LIN {X 0,Y 192.348,Z 460.48,A -85,B 0,C 180,E1 -21860.529,E2 -21860.529} C_VEL
LIN {X 0,Y 193.959,Z 454.471,A -85,B 0,C 180,E1 -21863.761,E2 -21863.761} C_VEL
LIN {X 0,Y 196.232,Z 446.608,A -85,B 0,C 180,E1 -21867.025,E2 -21867.025} C_VEL
LIN {X 0,Y 198.774,Z 437.463,A -85,B 0,C 180,E1 -21870.002,E2 -21870.002} C_VEL
LIN {X 0,Y 201.367,Z 427.594,A -85,B 0,C 180,E1 -21872.502,E2 -21872.502} C_VEL
LIN {X 0,Y 204.103,Z 416.202,A -85,B 0,C 180,E1 -21874.764,E2 -21874.764} C_VEL
LIN {X 0,Y 206.217,Z 405.922,A -85,B 0,C 180,E1 -21876.361,E2 -21876.361} C_VEL
LIN {X 0,Y 208.161,Z 394.258,A -85,B 0,C 180,E1 -21877.763,E2 -21877.763} C_VEL
LIN {X 0,Y 209.919,Z 381.041,A -85,B 0,C 180,E1 -21878.909,E2 -21878.909} C_VEL
LIN {X 0,Y 211.115,Z 368.346,A -85,B 0,C 180,E1 -21879.633,E2 -21879.633} C_VEL
LIN {X 0,Y 213.846,Z 309.716,A -85,B 0,C 180,E1 -21881.608,E2 -21881.608} C_VEL
LIN {X 0,Y 206.528,Z 290.704,A -85,B 0,C 180,E1 -21883.594,E2 -21883.594} C_VEL
LIN {X 0,Y 198.591,Z 273.838,A -85,B 0,C 180,E1 -21885.769,E2 -21885.769} C_VEL
LIN {X 0,Y 194.153,Z 266.401,A -85,B 0,C 180,E1 -21886.995,E2 -21886.995} C_VEL
LIN {X 0,Y 192.896,Z 263.787,A -85,B 0,C 180,E1 -21887.477,E2 -21887.477} C_VEL
LIN {X 0,Y 192.743,Z 263.034,A -85,B 0,C 180,E1 -21887.926,E2 -21887.926} C_VEL
LIN {X 0,Y 192.652,Z 262.975,A -85,B 0,C 180,E1 -21893.66,E2 -21893.66} C_VEL
LIN {X 0,Y 192.577,Z 262.979,A -85,B 0,C 180,E1 -21898.87,E2 -21898.87} C_VEL
LIN {X 0,Y 192.571,Z 262.99,A -85,B 0,C 180,E1 -21903.193,E2 -21903.193} C_VEL
LIN {X 0,Y 192.521,Z 263.004,A -85,B 0,C 180,E1 -21908.361,E2 -21908.361} C_VEL
LIN {X 0,Y 192.465,Z 262.982,A -85,B 0,C 180,E1 -21913.1,E2 -21913.1} C_VEL
LIN {X 0,Y 192.469,Z 263.011,A -85,B 0,C 180,E1 -21916.913,E2 -21916.913} C_VEL
LIN {X 0,Y 192.527,Z 262.965,A -85,B 0,C 180,E1 -21921.653,E2 -21921.653} C_VEL
LIN {X 0,Y 192.583,Z 262.994,A -85,B 0,C 180,E1 -21926.821,E2 -21926.821} C_VEL
LIN {X 0,Y 192.601,Z 262.948,A -85,B 0,C 180,E1 -21931.691,E2 -21931.691} C_VEL
LIN {X 0,Y 192.653,Z 262.986,A -85,B 0,C 180,E1 -21936.35,E2 -21936.35} C_VEL
LIN {X 0,Y 192.692,Z 262.933,A -85,B 0,C 180,E1 -21941.498,E2 -21941.498} C_VEL
LIN {X 0,Y 192.739,Z 262.95,A -85,B 0,C 180,E1 -21945.22,E2 -21945.22} C_VEL
LIN {X 0,Y 192.946,Z 262.944,A -85,B 0,C 180,E1 -21949.574,E2 -21949.574} C_VEL
LIN {X 0,Y 192.965,Z 262.897,A -85,B 0,C 180,E1 -21953.735,E2 -21953.735} C_VEL
LIN {X 0,Y 193.232,Z 262.904,A -85,B 0,C 180,E1 -21957.923,E2 -21957.923} C_VEL
LIN {X 0,Y 193.417,Z 262.891,A -85,B 0,C 180,E1 -21960.007,E2 -21960.007} C_VEL
LIN {X 0,Y 192.937,Z 262.907,A -85,B 0,C 180,E1 -21964.185,E2 -21964.185} C_VEL
LIN {X 0,Y 193.039,Z 262.926,A -85,B 0,C 180,E1 -21968.381,E2 -21968.381} C_VEL
LIN {X 0,Y 192.805,Z 262.955,A -85,B 0,C 180,E1 -21972.64,E2 -21972.64} C_VEL
LIN {X 0,Y 192.732,Z 262.949,A -85,B 0,C 180,E1 -21976.968,E2 -21976.968} C_VEL
LIN {X 0,Y 192.62,Z 262.984,A -85,B 0,C 180,E1 -21981.406,E2 -21981.406} C_VEL
LIN {X 0,Y 192.652,Z 262.956,A -85,B 0,C 180,E1 -21984.213,E2 -21984.213} C_VEL
LIN {X 0,Y 192.616,Z 262.987,A -85,B 0,C 180,E1 -21988.87,E2 -21988.87} C_VEL
LIN {X 0,Y 192.609,Z 262.983,A -85,B 0,C 180,E1 -21993.191,E2 -21993.191} C_VEL
LIN {X 0,Y 192.557,Z 262.985,A -85,B 0,C 180,E1 -21998.358,E2 -21998.358} C_VEL
LIN {X 0,Y 192.5,Z 262.993,A -85,B 0,C 180,E1 -22003.096,E2 -22003.096} C_VEL
LIN {X 0,Y 192.598,Z 263.215,A -85,B 0,C 180,E1 -22007.845,E2 -22007.845} C_VEL
LIN {X 0,Y 193.472,Z 266.459,A -85,B 0,C 180,E1 -22009.626,E2 -22009.626} C_VEL
LIN {X 0,Y 199.825,Z 279.379,A -85,B 0,C 180,E1 -22011.546,E2 -22011.546} C_VEL
LIN {X 0,Y 207.254,Z 296.355,A -85,B 0,C 180,E1 -22013.6,E2 -22013.6} C_VEL
LIN {X 0,Y 212.281,Z 309.796,A -85,B 0,C 180,E1 -22014.982,E2 -22014.982} C_VEL
LIN {X 0,Y 213.59,Z 320.418,A -85,B 0,C 180,E1 -22015.614,E2 -22015.614} C_VEL
LIN {X 0,Y 213.361,Z 326.003,A -85,B 0,C 180,E1 -22015.803,E2 -22015.803} C_VEL
LIN {X 0,Y 212.523,Z 331.839,A -85,B 0,C 180,E1 -22015.909,E2 -22015.909} C_VEL
LIN {X 0,Y 206.506,Z 350.757,A -85,B 0,C 180,E1 -22015.752,E2 -22015.752} C_VEL
LIN {X 0,Y 205.647,Z 356.594,A -85,B 0,C 180,E1 -22015.859,E2 -22015.859} C_VEL
LIN {X 0,Y 204.571,Z 375.827,A -85,B 0,C 180,E1 -22016.577,E2 -22016.577} C_VEL
LIN {X 0,Y 203.127,Z 389.153,A -85,B 0,C 180,E1 -22017.42,E2 -22017.42} C_VEL
LIN {X 0,Y 201.302,Z 401.297,A -85,B 0,C 180,E1 -22018.565,E2 -22018.565} C_VEL
LIN {X 0,Y 199.045,Z 413.08,A -85,B 0,C 180,E1 -22020.082,E2 -22020.082} C_VEL
LIN {X 0,Y 196.366,Z 424.446,A -85,B 0,C 180,E1 -22021.98,E2 -22021.98} C_VEL
LIN {X 0,Y 193.702,Z 434.702,A -85,B 0,C 180,E1 -22024.188,E2 -22024.188} C_VEL
LIN {X 0,Y 191.305,Z 443.865,A -85,B 0,C 180,E1 -22026.711,E2 -22026.711} C_VEL
LIN {X 0,Y 189.106,Z 451.549,A -85,B 0,C 180,E1 -22029.324,E2 -22029.324} C_VEL
LIN {X 0,Y 186.872,Z 458.998,A -85,B 0,C 180,E1 -22032.488,E2 -22032.488} C_VEL
LIN {X 0,Y 185.181,Z 464.964,A -85,B 0,C 180,E1 -22035.717,E2 -22035.717} C_VEL
LIN {X 0,Y 184.066,Z 469.659,A -85,B 0,C 180,E1 -22038.992,E2 -22038.992} C_VEL
LIN {X 0,Y 183.347,Z 473.216,A -85,B 0,C 180,E1 -22042.288,E2 -22042.288} C_VEL
LIN {X 0,Y 183.036,Z 475.745,A -85,B 0,C 180,E1 -22045.594,E2 -22045.594} C_VEL
LIN {X 0,Y 183.009,Z 476.915,A -85,B 0,C 180,E1 -22047.797,E2 -22047.797} C_VEL
LIN {X 0,Y 183.075,Z 477.638,A -85,B 0,C 180,E1 -22049.998,E2 -22049.998} C_VEL
LIN {X 0,Y 183.005,Z 478.014,A -85,B 0,C 180,E1 -22053.051,E2 -22053.051} C_VEL
LIN {X 0,Y 183.246,Z 477.466,A -85,B 0,C 180,E1 -22056.605,E2 -22056.605} C_VEL
LIN {X 0,Y 184.182,Z 475.325,A -85,B 0,C 180,E1 -22060.997,E2 -22060.997} C_VEL
LIN {X 0,Y 185.46,Z 472.659,A -85,B 0,C 180,E1 -22064.258,E2 -22064.258} C_VEL
LIN {X 0,Y 187.222,Z 468.999,A -85,B 0,C 180,E1 -22067.474,E2 -22067.474} C_VEL
LIN {X 0,Y 189.73,Z 464.242,A -85,B 0,C 180,E1 -22070.602,E2 -22070.602} C_VEL
LIN {X 0,Y 192.578,Z 458.259,A -85,B 0,C 180,E1 -22073.666,E2 -22073.666} C_VEL
LIN {X 0,Y 196.004,Z 450.833,A -85,B 0,C 180,E1 -22076.626,E2 -22076.626} C_VEL
LIN {X 0,Y 199.205,Z 443.284,A -85,B 0,C 180,E1 -22079.017,E2 -22079.017} C_VEL
LIN {X 0,Y 202.927,Z 434.168,A -85,B 0,C 180,E1 -22081.296,E2 -22081.296} C_VEL
LIN {X 0,Y 206.482,Z 424.086,A -85,B 0,C 180,E1 -22083.286,E2 -22083.286} C_VEL
LIN {X 0,Y 209.868,Z 412.96,A -85,B 0,C 180,E1 -22084.991,E2 -22084.991} C_VEL
LIN {X 0,Y 213.01,Z 400.51,A -85,B 0,C 180,E1 -22086.431,E2 -22086.431} C_VEL
LIN {X 0,Y 215.37,Z 387.79,A -85,B 0,C 180,E1 -22087.5,E2 -22087.5} C_VEL
LIN {X 0,Y 217.245,Z 374.027,A -85,B 0,C 180,E1 -22088.245,E2 -22088.245} C_VEL
LIN {X 0,Y 220.362,Z 324.76,A -85,B 0,C 180,E1 -22089.87,E2 -22089.87} C_VEL
LIN {X 0,Y 215.479,Z 312.647,A -85,B 0,C 180,E1 -22091.831,E2 -22091.831} C_VEL
LIN {X 0,Y 209.653,Z 300.651,A -85,B 0,C 180,E1 -22094.301,E2 -22094.301} C_VEL
LIN {X 0,Y 203.954,Z 290.871,A -85,B 0,C 180,E1 -22096.917,E2 -22096.917} C_VEL
LIN {X 0,Y 200.622,Z 285.645,A -85,B 0,C 180,E1 -22098.58,E2 -22098.58} C_VEL
LIN {X 0,Y 198.031,Z 281.593,A -85,B 0,C 180,E1 -22099.979,E2 -22099.979} C_VEL
LIN {X 0,Y 194.419,Z 276.347,A -85,B 0,C 180,E1 -22102.075,E2 -22102.075} C_VEL
LIN {X 0,Y 189.987,Z 270.412,A -85,B 0,C 180,E1 -22105.007,E2 -22105.007} C_VEL
LIN {X 0,Y 186.281,Z 266.285,A -85,B 0,C 180,E1 -22107.778,E2 -22107.778} C_VEL
LIN {X 0,Y 185.636,Z 264.55,A -85,B 0,C 180,E1 -22108.623,E2 -22108.623} C_VEL
LIN {X 0,Y 185.545,Z 263.89,A -85,B 0,C 180,E1 -22109.554,E2 -22109.554} C_VEL
LIN {X 0,Y 185.583,Z 263.863,A -85,B 0,C 180,E1 -22115.375,E2 -22115.375} C_VEL
LIN {X 0,Y 185.658,Z 263.844,A -85,B 0,C 180,E1 -22121.142,E2 -22121.142} C_VEL
LIN {X 0,Y 185.681,Z 263.853,A -85,B 0,C 180,E1 -22124.629,E2 -22124.629} C_VEL
LIN {X 0,Y 185.886,Z 263.829,A -85,B 0,C 180,E1 -22129.412,E2 -22129.412} C_VEL
LIN {X 0,Y 185.925,Z 263.822,A -85,B 0,C 180,E1 -22133.481,E2 -22133.481} C_VEL
LIN {X 0,Y 186.167,Z 263.785,A -85,B 0,C 180,E1 -22137.829,E2 -22137.829} C_VEL
LIN {X 0,Y 186.366,Z 263.759,A -85,B 0,C 180,E1 -22139.993,E2 -22139.993} C_VEL
LIN {X 0,Y 185.918,Z 263.815,A -85,B 0,C 180,E1 -22146.504,E2 -22146.504} C_VEL
LIN {X 0,Y 185.957,Z 263.93,A -85,B 0,C 180,E1 -22148.995,E2 -22148.995} C_VEL
LIN {X 0,Y 186.632,Z 266.209,A -85,B 0,C 180,E1 -22149.707,E2 -22149.707} C_VEL
LIN {X 0,Y 188.658,Z 268.689,A -85,B 0,C 180,E1 -22151.271,E2 -22151.271} C_VEL
LIN {X 0,Y 190.328,Z 269.758,A -85,B 0,C 180,E1 -22152.386,E2 -22152.386} C_VEL
LIN {X 0,Y 192.014,Z 272.848,A -85,B 0,C 180,E1 -22153.62,E2 -22153.62} C_VEL
LIN {X 0,Y 194.475,Z 275.239,A -85,B 0,C 180,E1 -22155.114,E2 -22155.114} C_VEL
LIN {X 0,Y 196.797,Z 278.656,A -85,B 0,C 180,E1 -22156.494,E2 -22156.494} C_VEL
LIN {X 0,Y 198.411,Z 280.537,A -85,B 0,C 180,E1 -22157.366,E2 -22157.366} C_VEL
LIN {X 0,Y 202.199,Z 285.744,A -85,B 0,C 180,E1 -22159.318,E2 -22159.318} C_VEL
LIN {X 0,Y 207.313,Z 293.923,A -85,B 0,C 180,E1 -22161.756,E2 -22161.756} C_VEL
LIN {X 0,Y 213.612,Z 305.557,A -85,B 0,C 180,E1 -22164.477,E2 -22164.477} C_VEL
LIN {X 0,Y 218.814,Z 316.781,A -85,B 0,C 180,E1 -22166.57,E2 -22166.57} C_VEL
LIN {X 0,Y 220.593,Z 321.576,A -85,B 0,C 180,E1 -22167.281,E2 -22167.281} C_VEL
LIN {X 0,Y 217.359,Z 370.033,A -85,B 0,C 180,E1 -22168.846,E2 -22168.846} C_VEL
LIN {X 0,Y 215.632,Z 383.142,A -85,B 0,C 180,E1 -22169.567,E2 -22169.567} C_VEL
LIN {X 0,Y 213.37,Z 395.759,A -85,B 0,C 180,E1 -22170.63,E2 -22170.63} C_VEL
LIN {X 0,Y 210.697,Z 407.132,A -85,B 0,C 180,E1 -22171.946,E2 -22171.946} C_VEL
LIN {X 0,Y 207.136,Z 419.18,A -85,B 0,C 180,E1 -22173.774,E2 -22173.774} C_VEL
LIN {X 0,Y 203.321,Z 430.218,A -85,B 0,C 180,E1 -22175.979,E2 -22175.979} C_VEL
LIN {X 0,Y 199.518,Z 439.625,A -85,B 0,C 180,E1 -22178.398,E2 -22178.398} C_VEL
LIN {X 0,Y 195.86,Z 447.893,A -85,B 0,C 180,E1 -22181.105,E2 -22181.105} C_VEL
LIN {X 0,Y 192.849,Z 454.373,A -85,B 0,C 180,E1 -22183.81,E2 -22183.81} C_VEL
LIN {X 0,Y 189.997,Z 460.083,A -85,B 0,C 180,E1 -22186.821,E2 -22186.821} C_VEL
LIN {X 0,Y 187.356,Z 465.195,A -85,B 0,C 180,E1 -22190.383,E2 -22190.383} C_VEL
LIN {X 0,Y 185.35,Z 468.908,A -85,B 0,C 180,E1 -22194.007,E2 -22194.007} C_VEL
LIN {X 0,Y 183.967,Z 471.385,A -85,B 0,C 180,E1 -22197.67,E2 -22197.67} C_VEL
LIN {X 0,Y 183.294,Z 472.403,A -85,B 0,C 180,E1 -22200.105,E2 -22200.105} C_VEL
LIN {X 0,Y 182.851,Z 472.92,A -85,B 0,C 180,E1 -22202.536,E2 -22202.536} C_VEL
LIN {X 0,Y 182.576,Z 472.942,A -85,B 0,C 180,E1 -22204.951,E2 -22204.951} C_VEL
LIN {X 0,Y 182.55,Z 472.492,A -85,B 0,C 180,E1 -22207.491,E2 -22207.491} C_VEL
LIN {X 0,Y 182.615,Z 471.614,A -85,B 0,C 180,E1 -22209.737,E2 -22209.737} C_VEL
LIN {X 0,Y 183.156,Z 469.145,A -85,B 0,C 180,E1 -22213.563,E2 -22213.563} C_VEL
LIN {X 0,Y 183.903,Z 466.084,A -85,B 0,C 180,E1 -22216.746,E2 -22216.746} C_VEL
LIN {X 0,Y 185.212,Z 461.057,A -85,B 0,C 180,E1 -22220.549,E2 -22220.549} C_VEL
LIN {X 0,Y 186.949,Z 454.874,A -85,B 0,C 180,E1 -22224.068,E2 -22224.068} C_VEL
LIN {X 0,Y 189.194,Z 447.371,A -85,B 0,C 180,E1 -22227.34,E2 -22227.34} C_VEL
LIN {X 0,Y 191.913,Z 438.025,A -85,B 0,C 180,E1 -22230.526,E2 -22230.526} C_VEL
LIN {X 0,Y 194.594,Z 428.288,A -85,B 0,C 180,E1 -22233.107,E2 -22233.107} C_VEL
LIN {X 0,Y 197.278,Z 417.628,A -85,B 0,C 180,E1 -22235.324,E2 -22235.324} C_VEL
LIN {X 0,Y 199.626,Z 406.893,A -85,B 0,C 180,E1 -22237.08,E2 -22237.08} C_VEL
LIN {X 0,Y 201.807,Z 394.435,A -85,B 0,C 180,E1 -22238.639,E2 -22238.639} C_VEL
LIN {X 0,Y 203.618,Z 381.26,A -85,B 0,C 180,E1 -22239.814,E2 -22239.814} C_VEL
LIN {X 0,Y 204.862,Z 368.565,A -85,B 0,C 180,E1 -22240.559,E2 -22240.559} C_VEL
LIN {X 0,Y 207.706,Z 311.757,A -85,B 0,C 180,E1 -22242.509,E2 -22242.509} C_VEL
LIN {X 0,Y 201.093,Z 294.261,A -85,B 0,C 180,E1 -22244.394,E2 -22244.394} C_VEL
LIN {X 0,Y 193.716,Z 278.349,A -85,B 0,C 180,E1 -22246.526,E2 -22246.526} C_VEL
LIN {X 0,Y 187.389,Z 267.629,A -85,B 0,C 180,E1 -22248.373,E2 -22248.373} C_VEL
LIN {X 0,Y 185.884,Z 265.014,A -85,B 0,C 180,E1 -22248.897,E2 -22248.897} C_VEL
LIN {X 0,Y 185.611,Z 263.942,A -85,B 0,C 180,E1 -22249.425,E2 -22249.425} C_VEL
LIN {X 0,Y 185.553,Z 263.859,A -85,B 0,C 180,E1 -22254.651,E2 -22254.651} C_VEL
LIN {X 0,Y 185.52,Z 263.857,A -85,B 0,C 180,E1 -22259.505,E2 -22259.505} C_VEL
LIN {X 0,Y 185.475,Z 263.859,A -85,B 0,C 180,E1 -22264.639,E2 -22264.639} C_VEL
LIN {X 0,Y 185.479,Z 263.871,A -85,B 0,C 180,E1 -22267.321,E2 -22267.321} C_VEL
LIN {X 0,Y 185.441,Z 263.868,A -85,B 0,C 180,E1 -22270.728,E2 -22270.728} C_VEL
LIN {X 0,Y 185.439,Z 263.885,A -85,B 0,C 180,E1 -22276.064,E2 -22276.064} C_VEL
LIN {X 0,Y 185.441,Z 263.853,A -85,B 0,C 180,E1 -22279.899,E2 -22279.899} C_VEL
LIN {X 0,Y 185.487,Z 263.848,A -85,B 0,C 180,E1 -22282.722,E2 -22282.722} C_VEL
LIN {X 0,Y 185.519,Z 263.863,A -85,B 0,C 180,E1 -22287.98,E2 -22287.98} C_VEL
LIN {X 0,Y 185.481,Z 263.843,A -85,B 0,C 180,E1 -22292.965,E2 -22292.965} C_VEL
LIN {X 0,Y 185.55,Z 263.868,A -85,B 0,C 180,E1 -22297.752,E2 -22297.752} C_VEL
LIN {X 0,Y 185.651,Z 263.806,A -85,B 0,C 180,E1 -22302.38,E2 -22302.38} C_VEL
LIN {X 0,Y 185.718,Z 263.846,A -85,B 0,C 180,E1 -22306.884,E2 -22306.884} C_VEL
LIN {X 0,Y 185.974,Z 263.792,A -85,B 0,C 180,E1 -22311.314,E2 -22311.314} C_VEL
LIN {X 0,Y 186.178,Z 263.782,A -85,B 0,C 180,E1 -22317.844,E2 -22317.844} C_VEL
LIN {X 0,Y 186.383,Z 263.767,A -85,B 0,C 180,E1 -22320.007,E2 -22320.007} C_VEL
LIN {X 0,Y 185.886,Z 263.784,A -85,B 0,C 180,E1 -22324.344,E2 -22324.344} C_VEL
LIN {X 0,Y 185.987,Z 263.807,A -85,B 0,C 180,E1 -22328.701,E2 -22328.701} C_VEL
LIN {X 0,Y 185.73,Z 263.827,A -85,B 0,C 180,E1 -22333.13,E2 -22333.13} C_VEL
LIN {X 0,Y 185.668,Z 263.837,A -85,B 0,C 180,E1 -22337.634,E2 -22337.634} C_VEL
LIN {X 0,Y 185.583,Z 263.847,A -85,B 0,C 180,E1 -22342.26,E2 -22342.26} C_VEL
LIN {X 0,Y 185.591,Z 263.836,A -85,B 0,C 180,E1 -22344.651,E2 -22344.651} C_VEL
LIN {X 0,Y 185.558,Z 263.859,A -85,B 0,C 180,E1 -22349.504,E2 -22349.504} C_VEL
LIN {X 0,Y 185.512,Z 263.878,A -85,B 0,C 180,E1 -22354.637,E2 -22354.637} C_VEL
LIN {X 0,Y 185.515,Z 263.859,A -85,B 0,C 180,E1 -22357.319,E2 -22357.319} C_VEL
LIN {X 0,Y 185.477,Z 263.878,A -85,B 0,C 180,E1 -22360.725,E2 -22360.725} C_VEL
LIN {X 0,Y 185.472,Z 263.875,A -85,B 0,C 180,E1 -22366.06,E2 -22366.06} C_VEL
LIN {X 0,Y 185.506,Z 264.159,A -85,B 0,C 180,E1 -22366.798,E2 -22366.798} C_VEL
LIN {X 0,Y 186.126,Z 266.335,A -85,B 0,C 180,E1 -22368.038,E2 -22368.038} C_VEL
LIN {X 0,Y 191.726,Z 277.331,A -85,B 0,C 180,E1 -22369.846,E2 -22369.846} C_VEL
LIN {X 0,Y 198.232,Z 291.3,A -85,B 0,C 180,E1 -22371.777,E2 -22371.777} C_VEL
LIN {X 0,Y 205.091,Z 308.581,A -85,B 0,C 180,E1 -22373.751,E2 -22373.751} C_VEL
LIN {X 0,Y 206.461,Z 313.037,A -85,B 0,C 180,E1 -22374.17,E2 -22374.17} C_VEL
LIN {X 0,Y 207.432,Z 320.508,A -85,B 0,C 180,E1 -22374.644,E2 -22374.644} C_VEL
LIN {X 0,Y 205.647,Z 356.594,A -85,B 0,C 180,E1 -22375.859,E2 -22375.859} C_VEL
LIN {X 0,Y 204.788,Z 362.434,A -85,B 0,C 180,E1 -22375.961,E2 -22375.961} C_VEL
LIN {X 0,Y 201.711,Z 371.88,A -85,B 0,C 180,E1 -22375.904,E2 -22375.904} C_VEL
LIN {X 0,Y 198.41,Z 381.229,A -85,B 0,C 180,E1 -22375.994,E2 -22375.994} C_VEL
LIN {X 0,Y 197.195,Z 386.914,A -85,B 0,C 180,E1 -22376.307,E2 -22376.307} C_VEL
LIN {X 0,Y 195.213,Z 399.691,A -85,B 0,C 180,E1 -22377.466,E2 -22377.466} C_VEL
LIN {X 0,Y 192.847,Z 411.869,A -85,B 0,C 180,E1 -22379.017,E2 -22379.017} C_VEL
LIN {X 0,Y 190.11,Z 423.447,A -85,B 0,C 180,E1 -22380.972,E2 -22380.972} C_VEL
LIN {X 0,Y 187.346,Z 433.892,A -85,B 0,C 180,E1 -22383.244,E2 -22383.244} C_VEL
LIN {X 0,Y 184.542,Z 443.958,A -85,B 0,C 180,E1 -22386.079,E2 -22386.079} C_VEL
LIN {X 0,Y 181.993,Z 452.35,A -85,B 0,C 180,E1 -22389.07,E2 -22389.07} C_VEL
LIN {X 0,Y 179.758,Z 459.645,A -85,B 0,C 180,E1 -22392.36,E2 -22392.36} C_VEL
LIN {X 0,Y 178.252,Z 464.552,A -85,B 0,C 180,E1 -22395.149,E2 -22395.149} C_VEL
LIN {X 0,Y 177.063,Z 469.315,A -85,B 0,C 180,E1 -22398.551,E2 -22398.551} C_VEL
LIN {X 0,Y 176.298,Z 472.935,A -85,B 0,C 180,E1 -22401.978,E2 -22401.978} C_VEL
LIN {X 0,Y 175.959,Z 475.522,A -85,B 0,C 180,E1 -22405.416,E2 -22405.416} C_VEL
LIN {X 0,Y 175.906,Z 476.732,A -85,B 0,C 180,E1 -22407.708,E2 -22407.708} C_VEL
LIN {X 0,Y 175.987,Z 477.498,A -85,B 0,C 180,E1 -22409.998,E2 -22409.998} C_VEL
LIN {X 0,Y 175.928,Z 477.886,A -85,B 0,C 180,E1 -22412.803,E2 -22412.803} C_VEL
LIN {X 0,Y 176.175,Z 477.416,A -85,B 0,C 180,E1 -22416.871,E2 -22416.871} C_VEL
LIN {X 0,Y 176.596,Z 476.594,A -85,B 0,C 180,E1 -22419.158,E2 -22419.158} C_VEL
LIN {X 0,Y 178.045,Z 473.723,A -85,B 0,C 180,E1 -22423.698,E2 -22423.698} C_VEL
LIN {X 0,Y 179.749,Z 470.458,A -85,B 0,C 180,E1 -22427.05,E2 -22427.05} C_VEL
LIN {X 0,Y 182.157,Z 466.145,A -85,B 0,C 180,E1 -22430.316,E2 -22430.316} C_VEL
LIN {X 0,Y 185.102,Z 460.672,A -85,B 0,C 180,E1 -22433.493,E2 -22433.493} C_VEL
LIN {X 0,Y 188.397,Z 453.879,A -85,B 0,C 180,E1 -22436.591,E2 -22436.591} C_VEL
LIN {X 0,Y 192.363,Z 445.431,A -85,B 0,C 180,E1 -22439.55,E2 -22439.55} C_VEL
LIN {X 0,Y 196.146,Z 436.77,A -85,B 0,C 180,E1 -22441.902,E2 -22441.902} C_VEL
LIN {X 0,Y 200.17,Z 426.159,A -85,B 0,C 180,E1 -22444.175,E2 -22444.175} C_VEL
LIN {X 0,Y 203.698,Z 415.621,A -85,B 0,C 180,E1 -22445.909,E2 -22445.909} C_VEL
LIN {X 0,Y 206.919,Z 403.903,A -85,B 0,C 180,E1 -22447.379,E2 -22447.379} C_VEL
LIN {X 0,Y 209.747,Z 390.582,A -85,B 0,C 180,E1 -22448.611,E2 -22448.611} C_VEL
LIN {X 0,Y 211.79,Z 377.37,A -85,B 0,C 180,E1 -22449.415,E2 -22449.415} C_VEL
LIN {X 0,Y 213.149,Z 360.665,A -85,B 0,C 180,E1 -22450.04,E2 -22450.04} C_VEL
LIN {X 0,Y 215.281,Z 326.927,A -85,B 0,C 180,E1 -22451.152,E2 -22451.152} C_VEL
LIN {X 0,Y 210.459,Z 315.083,A -85,B 0,C 180,E1 -22453.237,E2 -22453.237} C_VEL
LIN {X 0,Y 205.726,Z 305.156,A -85,B 0,C 180,E1 -22455.389,E2 -22455.389} C_VEL
LIN {X 0,Y 200.283,Z 295.554,A -85,B 0,C 180,E1 -22458.067,E2 -22458.067} C_VEL
LIN {X 0,Y 195.288,Z 287.454,A -85,B 0,C 180,E1 -22460.825,E2 -22460.825} C_VEL
LIN {X 0,Y 191.602,Z 282.079,A -85,B 0,C 180,E1 -22463.084,E2 -22463.084} C_VEL
LIN {X 0,Y 187.916,Z 276.824,A -85,B 0,C 180,E1 -22465.685,E2 -22465.685} C_VEL
LIN {X 0,Y 184.285,Z 272.69,A -85,B 0,C 180,E1 -22468.526,E2 -22468.526} C_VEL
LIN {X 0,Y 183.158,Z 270.59,A -85,B 0,C 180,E1 -22469.593,E2 -22469.593} C_VEL
LIN {X 0,Y 180.214,Z 268.613,A -85,B 0,C 180,E1 -22472.405,E2 -22472.405} C_VEL
LIN {X 0,Y 178.801,Z 266.137,A -85,B 0,C 180,E1 -22474.218,E2 -22474.218} C_VEL
LIN {X 0,Y 178.518,Z 264.751,A -85,B 0,C 180,E1 -22474.882,E2 -22474.882} C_VEL
LIN {X 0,Y 178.61,Z 264.723,A -85,B 0,C 180,E1 -22480.79,E2 -22480.79} C_VEL
LIN {X 0,Y 178.647,Z 264.715,A -85,B 0,C 180,E1 -22486.34,E2 -22486.34} C_VEL
LIN {X 0,Y 178.902,Z 264.684,A -85,B 0,C 180,E1 -22490.952,E2 -22490.952} C_VEL
LIN {X 0,Y 179.114,Z 264.663,A -85,B 0,C 180,E1 -22497.744,E2 -22497.744} C_VEL
LIN {X 0,Y 179.331,Z 264.635,A -85,B 0,C 180,E1 -22499.992,E2 -22499.992} C_VEL
LIN {X 0,Y 178.984,Z 264.743,A -85,B 0,C 180,E1 -22503.017,E2 -22503.017} C_VEL
LIN {X 0,Y 179.528,Z 266.936,A -85,B 0,C 180,E1 -22503.92,E2 -22503.92} C_VEL
LIN {X 0,Y 181.067,Z 269.022,A -85,B 0,C 180,E1 -22505.7,E2 -22505.7} C_VEL
LIN {X 0,Y 183.808,Z 270.727,A -85,B 0,C 180,E1 -22508.167,E2 -22508.167} C_VEL
LIN {X 0,Y 185.166,Z 273.471,A -85,B 0,C 180,E1 -22509.432,E2 -22509.432} C_VEL
LIN {X 0,Y 187.543,Z 275.818,A -85,B 0,C 180,E1 -22511.236,E2 -22511.236} C_VEL
LIN {X 0,Y 188.296,Z 276.695,A -85,B 0,C 180,E1 -22511.787,E2 -22511.787} C_VEL
LIN {X 0,Y 190.594,Z 280.073,A -85,B 0,C 180,E1 -22513.435,E2 -22513.435} C_VEL
LIN {X 0,Y 192.139,Z 281.747,A -85,B 0,C 180,E1 -22514.421,E2 -22514.421} C_VEL
LIN {X 0,Y 195.003,Z 285.554,A -85,B 0,C 180,E1 -22516.144,E2 -22516.144} C_VEL
LIN {X 0,Y 199.362,Z 291.728,A -85,B 0,C 180,E1 -22518.549,E2 -22518.549} C_VEL
LIN {X 0,Y 204.327,Z 299.961,A -85,B 0,C 180,E1 -22521.031,E2 -22521.031} C_VEL
LIN {X 0,Y 210.344,Z 311.56,A -85,B 0,C 180,E1 -22523.776,E2 -22523.776} C_VEL
LIN {X 0,Y 215.292,Z 322.961,A -85,B 0,C 180,E1 -22525.892,E2 -22525.892} C_VEL
LIN {X 0,Y 215.532,Z 323.961,A -85,B 0,C 180,E1 -22526.013,E2 -22526.013} C_VEL
LIN {X 0,Y 212.28,Z 370.287,A -85,B 0,C 180,E1 -22527.53,E2 -22527.53} C_VEL
LIN {X 0,Y 210.538,Z 383.029,A -85,B 0,C 180,E1 -22528.235,E2 -22528.235} C_VEL
LIN {X 0,Y 208.106,Z 396.067,A -85,B 0,C 180,E1 -22529.345,E2 -22529.345} C_VEL
LIN {X 0,Y 205.309,Z 407.418,A -85,B 0,C 180,E1 -22530.68,E2 -22530.68} C_VEL
LIN {X 0,Y 201.848,Z 418.676,A -85,B 0,C 180,E1 -22532.402,E2 -22532.402} C_VEL
LIN {X 0,Y 198.307,Z 428.557,A -85,B 0,C 180,E1 -22534.346,E2 -22534.346} C_VEL
LIN {X 0,Y 194.636,Z 437.462,A -85,B 0,C 180,E1 -22536.546,E2 -22536.546} C_VEL
LIN {X 0,Y 190.683,Z 446.132,A -85,B 0,C 180,E1 -22539.289,E2 -22539.289} C_VEL
LIN {X 0,Y 187.145,Z 453.297,A -85,B 0,C 180,E1 -22542.204,E2 -22542.204} C_VEL
LIN {X 0,Y 184.213,Z 458.915,A -85,B 0,C 180,E1 -22545.109,E2 -22545.109} C_VEL
LIN {X 0,Y 181.229,Z 464.327,A -85,B 0,C 180,E1 -22548.76,E2 -22548.76} C_VEL
LIN {X 0,Y 179.427,Z 467.458,A -85,B 0,C 180,E1 -22551.556,E2 -22551.556} C_VEL
LIN {X 0,Y 178.303,Z 469.377,A -85,B 0,C 180,E1 -22553.758,E2 -22553.758} C_VEL
LIN {X 0,Y 177.261,Z 471.122,A -85,B 0,C 180,E1 -22556.35,E2 -22556.35} C_VEL
LIN {X 0,Y 176.485,Z 472.232,A -85,B 0,C 180,E1 -22558.825,E2 -22558.825} C_VEL
LIN {X 0,Y 175.911,Z 472.934,A -85,B 0,C 180,E1 -22561.495,E2 -22561.495} C_VEL
LIN {X 0,Y 175.558,Z 473.103,A -85,B 0,C 180,E1 -22563.876,E2 -22563.876} C_VEL
LIN {X 0,Y 175.44,Z 472.637,A -85,B 0,C 180,E1 -22567.102,E2 -22567.102} C_VEL
LIN {X 0,Y 175.676,Z 470.829,A -85,B 0,C 180,E1 -22571.337,E2 -22571.337} C_VEL
LIN {X 0,Y 176.35,Z 468.111,A -85,B 0,C 180,E1 -22574.989,E2 -22574.989} C_VEL
LIN {X 0,Y 177.355,Z 464.295,A -85,B 0,C 180,E1 -22578.574,E2 -22578.574} C_VEL
LIN {X 0,Y 178.76,Z 459.285,A -85,B 0,C 180,E1 -22582.093,E2 -22582.093} C_VEL
LIN {X 0,Y 180.666,Z 452.931,A -85,B 0,C 180,E1 -22585.54,E2 -22585.54} C_VEL
LIN {X 0,Y 182.984,Z 445.446,A -85,B 0,C 180,E1 -22588.727,E2 -22588.727} C_VEL
LIN {X 0,Y 185.568,Z 436.782,A -85,B 0,C 180,E1 -22591.629,E2 -22591.629} C_VEL
LIN {X 0,Y 188.469,Z 426.705,A -85,B 0,C 180,E1 -22594.279,E2 -22594.279} C_VEL
LIN {X 0,Y 191.212,Z 416.039,A -85,B 0,C 180,E1 -22596.485,E2 -22596.485} C_VEL
LIN {X 0,Y 193.758,Z 404.357,A -85,B 0,C 180,E1 -22598.344,E2 -22598.344} C_VEL
LIN {X 0,Y 195.838,Z 392.217,A -85,B 0,C 180,E1 -22599.816,E2 -22599.816} C_VEL
LIN {X 0,Y 197.564,Z 379.761,A -85,B 0,C 180,E1 -22600.895,E2 -22600.895} C_VEL
LIN {X 0,Y 198.781,Z 367,A -85,B 0,C 180,E1 -22601.602,E2 -22601.602} C_VEL
LIN {X 0,Y 201.601,Z 313.592,A -85,B 0,C 180,E1 -22603.462,E2 -22603.462} C_VEL
LIN {X 0,Y 195.268,Z 296.731,A -85,B 0,C 180,E1 -22605.37,E2 -22605.37} C_VEL
LIN {X 0,Y 188.275,Z 281.78,A -85,B 0,C 180,E1 -22607.492,E2 -22607.492} C_VEL
LIN {X 0,Y 182.013,Z 271.299,A -85,B 0,C 180,E1 -22609.411,E2 -22609.411} C_VEL
LIN {X 0,Y 180.337,Z 268.639,A -85,B 0,C 180,E1 -22609.948,E2 -22609.948} C_VEL
LIN {X 0,Y 178.774,Z 265.941,A -85,B 0,C 180,E1 -22610.52,E2 -22610.52} C_VEL
LIN {X 0,Y 178.505,Z 264.844,A -85,B 0,C 180,E1 -22611.057,E2 -22611.057} C_VEL
LIN {X 0,Y 178.462,Z 264.748,A -85,B 0,C 180,E1 -22615.672,E2 -22615.672} C_VEL
LIN {X 0,Y 178.437,Z 264.747,A -85,B 0,C 180,E1 -22620.801,E2 -22620.801} C_VEL
LIN {X 0,Y 178.46,Z 264.735,A -85,B 0,C 180,E1 -22624.224,E2 -22624.224} C_VEL
LIN {X 0,Y 178.367,Z 264.767,A -85,B 0,C 180,E1 -22629.084,E2 -22629.084} C_VEL
LIN {X 0,Y 178.374,Z 264.736,A -85,B 0,C 180,E1 -22632.054,E2 -22632.054} C_VEL
LIN {X 0,Y 178.374,Z 264.756,A -85,B 0,C 180,E1 -22635.173,E2 -22635.173} C_VEL
LIN {X 0,Y 178.382,Z 264.752,A -85,B 0,C 180,E1 -22638.469,E2 -22638.469} C_VEL
LIN {X 0,Y 178.406,Z 264.742,A -85,B 0,C 180,E1 -22643.79,E2 -22643.79} C_VEL
LIN {X 0,Y 178.472,Z 264.753,A -85,B 0,C 180,E1 -22646.554,E2 -22646.554} C_VEL
LIN {X 0,Y 178.412,Z 264.714,A -85,B 0,C 180,E1 -22651.8,E2 -22651.8} C_VEL
LIN {X 0,Y 178.463,Z 264.754,A -85,B 0,C 180,E1 -22656.818,E2 -22656.818} C_VEL
LIN {X 0,Y 178.606,Z 264.685,A -85,B 0,C 180,E1 -22661.66,E2 -22661.66} C_VEL
LIN {X 0,Y 178.644,Z 264.719,A -85,B 0,C 180,E1 -22666.355,E2 -22666.355} C_VEL
LIN {X 0,Y 178.905,Z 264.676,A -85,B 0,C 180,E1 -22670.967,E2 -22670.967} C_VEL
LIN {X 0,Y 179.126,Z 264.658,A -85,B 0,C 180,E1 -22677.759,E2 -22677.759} C_VEL
LIN {X 0,Y 179.348,Z 264.644,A -85,B 0,C 180,E1 -22680.008,E2 -22680.008} C_VEL
LIN {X 0,Y 178.835,Z 264.66,A -85,B 0,C 180,E1 -22684.515,E2 -22684.515} C_VEL
LIN {X 0,Y 178.917,Z 264.691,A -85,B 0,C 180,E1 -22689.047,E2 -22689.047} C_VEL
LIN {X 0,Y 178.656,Z 264.7,A -85,B 0,C 180,E1 -22693.66,E2 -22693.66} C_VEL
LIN {X 0,Y 178.602,Z 264.736,A -85,B 0,C 180,E1 -22699.192,E2 -22699.192} C_VEL
LIN {X 0,Y 178.529,Z 264.718,A -85,B 0,C 180,E1 -22705.116,E2 -22705.116} C_VEL
LIN {X 0,Y 178.474,Z 264.73,A -85,B 0,C 180,E1 -22710.799,E2 -22710.799} C_VEL
LIN {X 0,Y 178.497,Z 264.752,A -85,B 0,C 180,E1 -22714.222,E2 -22714.222} C_VEL
LIN {X 0,Y 178.403,Z 264.753,A -85,B 0,C 180,E1 -22719.081,E2 -22719.081} C_VEL
LIN {X 0,Y 178.409,Z 264.748,A -85,B 0,C 180,E1 -22722.051,E2 -22722.051} C_VEL
LIN {X 0,Y 178.436,Z 264.976,A -85,B 0,C 180,E1 -22725.561,E2 -22725.561} C_VEL
LIN {X 0,Y 178.85,Z 266.398,A -85,B 0,C 180,E1 -22726.335,E2 -22726.335} C_VEL
LIN {X 0,Y 184.343,Z 276.82,A -85,B 0,C 180,E1 -22728.238,E2 -22728.238} C_VEL
LIN {X 0,Y 190.525,Z 289.498,A -85,B 0,C 180,E1 -22730.175,E2 -22730.175} C_VEL
LIN {X 0,Y 198.176,Z 308.182,A -85,B 0,C 180,E1 -22732.522,E2 -22732.522} C_VEL
LIN {X 0,Y 200.525,Z 315.194,A -85,B 0,C 180,E1 -22733.251,E2 -22733.251} C_VEL
LIN {X 0,Y 201.307,Z 321.809,A -85,B 0,C 180,E1 -22733.674,E2 -22733.674} C_VEL
LIN {X 0,Y 198.468,Z 374.91,A -85,B 0,C 180,E1 -22735.563,E2 -22735.563} C_VEL
LIN {X 0,Y 197.195,Z 386.914,A -85,B 0,C 180,E1 -22736.307,E2 -22736.307} C_VEL
LIN {X 0,Y 196.369,Z 390.67,A -85,B 0,C 180,E1 -22736.552,E2 -22736.552} C_VEL
LIN {X 0,Y 193.461,Z 397.902,A -85,B 0,C 180,E1 -22736.96,E2 -22736.96} C_VEL
LIN {X 0,Y 187.79,Z 409.201,A -85,B 0,C 180,E1 -22737.809,E2 -22737.809} C_VEL
LIN {X 0,Y 185.73,Z 415.19,A -85,B 0,C 180,E1 -22738.609,E2 -22738.609} C_VEL
LIN {X 0,Y 182.858,Z 426.203,A -85,B 0,C 180,E1 -22740.655,E2 -22740.655} C_VEL
LIN {X 0,Y 180.337,Z 435.073,A -85,B 0,C 180,E1 -22742.746,E2 -22742.746} C_VEL
LIN {X 0,Y 177.762,Z 444.106,A -85,B 0,C 180,E1 -22745.427,E2 -22745.427} C_VEL
LIN {X 0,Y 175.366,Z 451.754,A -85,B 0,C 180,E1 -22748.239,E2 -22748.239} C_VEL
LIN {X 0,Y 172.955,Z 459.134,A -85,B 0,C 180,E1 -22751.642,E2 -22751.642} C_VEL
LIN {X 0,Y 171.352,Z 464.12,A -85,B 0,C 180,E1 -22754.536,E2 -22754.536} C_VEL
LIN {X 0,Y 170.087,Z 468.956,A -85,B 0,C 180,E1 -22758.075,E2 -22758.075} C_VEL
LIN {X 0,Y 169.242,Z 472.641,A -85,B 0,C 180,E1 -22761.641,E2 -22761.641} C_VEL
LIN {X 0,Y 168.878,Z 475.291,A -85,B 0,C 180,E1 -22765.224,E2 -22765.224} C_VEL
LIN {X 0,Y 168.804,Z 476.662,A -85,B 0,C 180,E1 -22767.895,E2 -22767.895} C_VEL
LIN {X 0,Y 168.885,Z 477.355,A -85,B 0,C 180,E1 -22769.998,E2 -22769.998} C_VEL
LIN {X 0,Y 168.836,Z 477.74,A -85,B 0,C 180,E1 -22772.384,E2 -22772.384} C_VEL
LIN {X 0,Y 169.13,Z 477.36,A -85,B 0,C 180,E1 -22777.159,E2 -22777.159} C_VEL
LIN {X 0,Y 169.567,Z 476.591,A -85,B 0,C 180,E1 -22779.541,E2 -22779.541} C_VEL
LIN {X 0,Y 171.144,Z 473.786,A -85,B 0,C 180,E1 -22784.262,E2 -22784.262} C_VEL
LIN {X 0,Y 172.97,Z 470.593,A -85,B 0,C 180,E1 -22787.74,E2 -22787.74} C_VEL
LIN {X 0,Y 175.52,Z 466.359,A -85,B 0,C 180,E1 -22791.121,E2 -22791.121} C_VEL
LIN {X 0,Y 179.1,Z 459.971,A -85,B 0,C 180,E1 -22794.948,E2 -22794.948} C_VEL
LIN {X 0,Y 182.751,Z 453.025,A -85,B 0,C 180,E1 -22798.103,E2 -22798.103} C_VEL
LIN {X 0,Y 186.974,Z 444.357,A -85,B 0,C 180,E1 -22801.118,E2 -22801.118} C_VEL
LIN {X 0,Y 191.016,Z 435.499,A -85,B 0,C 180,E1 -22803.494,E2 -22803.494} C_VEL
LIN {X 0,Y 195.331,Z 424.615,A -85,B 0,C 180,E1 -22805.778,E2 -22805.778} C_VEL
LIN {X 0,Y 198.999,Z 413.676,A -85,B 0,C 180,E1 -22807.53,E2 -22807.53} C_VEL
LIN {X 0,Y 202.385,Z 401.498,A -85,B 0,C 180,E1 -22809.004,E2 -22809.004} C_VEL
LIN {X 0,Y 205.064,Z 388.687,A -85,B 0,C 180,E1 -22810.144,E2 -22810.144} C_VEL
LIN {X 0,Y 207.126,Z 375.16,A -85,B 0,C 180,E1 -22810.911,E2 -22810.911} C_VEL
LIN {X 0,Y 209.371,Z 345.365,A -85,B 0,C 180,E1 -22811.935,E2 -22811.935} C_VEL
LIN {X 0,Y 210.346,Z 329.206,A -85,B 0,C 180,E1 -22812.504,E2 -22812.504} C_VEL
LIN {X 0,Y 206.129,Z 318.751,A -85,B 0,C 180,E1 -22814.452,E2 -22814.452} C_VEL
LIN {X 0,Y 201.967,Z 309.825,A -85,B 0,C 180,E1 -22816.494,E2 -22816.494} C_VEL
LIN {X 0,Y 196.996,Z 300.777,A -85,B 0,C 180,E1 -22819.095,E2 -22819.095} C_VEL
LIN {X 0,Y 192.566,Z 293.282,A -85,B 0,C 180,E1 -22821.716,E2 -22821.716} C_VEL
LIN {X 0,Y 189.241,Z 288.231,A -85,B 0,C 180,E1 -22823.882,E2 -22823.882} C_VEL
LIN {X 0,Y 185.547,Z 282.854,A -85,B 0,C 180,E1 -22826.628,E2 -22826.628} C_VEL
LIN {X 0,Y 182.274,Z 278.968,A -85,B 0,C 180,E1 -22829.35,E2 -22829.35} C_VEL
LIN {X 0,Y 181.388,Z 277.308,A -85,B 0,C 180,E1 -22830.252,E2 -22830.252} C_VEL
LIN {X 0,Y 178.601,Z 275.19,A -85,B 0,C 180,E1 -22833.086,E2 -22833.086} C_VEL
LIN {X 0,Y 177.069,Z 272.368,A -85,B 0,C 180,E1 -22835.196,E2 -22835.196} C_VEL
LIN {X 0,Y 176.743,Z 271.627,A -85,B 0,C 180,E1 -22835.712,E2 -22835.712} C_VEL
LIN {X 0,Y 173.723,Z 269.879,A -85,B 0,C 180,E1 -22840.752,E2 -22840.752} C_VEL
LIN {X 0,Y 172.168,Z 267.39,A -85,B 0,C 180,E1 -22848.421,E2 -22848.421} C_VEL
LIN {X 0,Y 172.429,Z 267.665,A -85,B 0,C 180,E1 -22851.496,E2 -22851.496} C_VEL
LIN {X 0,Y 177.13,Z 271.478,A -85,B 0,C 180,E1 -22861.981,E2 -22861.981} C_VEL
LIN {X 0,Y 178.597,Z 274.668,A -85,B 0,C 180,E1 -22864.082,E2 -22864.082} C_VEL
LIN {X 0,Y 181.07,Z 276.893,A -85,B 0,C 180,E1 -22866.679,E2 -22866.679} C_VEL
LIN {X 0,Y 181.957,Z 277.541,A -85,B 0,C 180,E1 -22867.482,E2 -22867.482} C_VEL
LIN {X 0,Y 183.859,Z 280.716,A -85,B 0,C 180,E1 -22869.259,E2 -22869.259} C_VEL
LIN {X 0,Y 186.117,Z 283.07,A -85,B 0,C 180,E1 -22871.013,E2 -22871.013} C_VEL
LIN {X 0,Y 188.676,Z 286.696,A -85,B 0,C 180,E1 -22872.906,E2 -22872.906} C_VEL
LIN {X 0,Y 189.923,Z 288.237,A -85,B 0,C 180,E1 -22873.75,E2 -22873.75} C_VEL
LIN {X 0,Y 193.428,Z 293.07,A -85,B 0,C 180,E1 -22875.941,E2 -22875.941} C_VEL
LIN {X 0,Y 196.726,Z 297.939,A -85,B 0,C 180,E1 -22877.832,E2 -22877.832} C_VEL
LIN {X 0,Y 201.208,Z 305.666,A -85,B 0,C 180,E1 -22880.199,E2 -22880.199} C_VEL
LIN {X 0,Y 206.931,Z 317.265,A -85,B 0,C 180,E1 -22882.98,E2 -22882.98} C_VEL
LIN {X 0,Y 210.599,Z 325.924,A -85,B 0,C 180,E1 -22884.64,E2 -22884.64} C_VEL
LIN {X 0,Y 207.39,Z 370.345,A -85,B 0,C 180,E1 -22886.13,E2 -22886.13} C_VEL
LIN {X 0,Y 205.552,Z 383.243,A -85,B 0,C 180,E1 -22886.85,E2 -22886.85} C_VEL
LIN {X 0,Y 203.213,Z 395.232,A -85,B 0,C 180,E1 -22887.868,E2 -22887.868} C_VEL
LIN {X 0,Y 200.43,Z 406.412,A -85,B 0,C 180,E1 -22889.166,E2 -22889.166} C_VEL
LIN {X 0,Y 197.109,Z 416.947,A -85,B 0,C 180,E1 -22890.737,E2 -22890.737} C_VEL
LIN {X 0,Y 193.26,Z 427.419,A -85,B 0,C 180,E1 -22892.763,E2 -22892.763} C_VEL
LIN {X 0,Y 189.098,Z 437.136,A -85,B 0,C 180,E1 -22895.153,E2 -22895.153} C_VEL
LIN {X 0,Y 184.91,Z 445.904,A -85,B 0,C 180,E1 -22897.943,E2 -22897.943} C_VEL
LIN {X 0,Y 180.586,Z 454.145,A -85,B 0,C 180,E1 -22901.41,E2 -22901.41} C_VEL
LIN {X 0,Y 177.423,Z 459.807,A -85,B 0,C 180,E1 -22904.523,E2 -22904.523} C_VEL
LIN {X 0,Y 174.312,Z 465.04,A -85,B 0,C 180,E1 -22908.301,E2 -22908.301} C_VEL
LIN {X 0,Y 171.902,Z 468.862,A -85,B 0,C 180,E1 -22912.177,E2 -22912.177} C_VEL
LIN {X 0,Y 170.436,Z 471.139,A -85,B 0,C 180,E1 -22915.542,E2 -22915.542} C_VEL
LIN {X 0,Y 169.083,Z 472.847,A -85,B 0,C 180,E1 -22920.083,E2 -22920.083} C_VEL
LIN {X 0,Y 168.587,Z 473.181,A -85,B 0,C 180,E1 -22922.708,E2 -22922.708} C_VEL
LIN {X 0,Y 168.328,Z 472.779,A -85,B 0,C 180,E1 -22926.689,E2 -22926.689} C_VEL
LIN {X 0,Y 168.472,Z 471.35,A -85,B 0,C 180,E1 -22930.507,E2 -22930.507} C_VEL
LIN {X 0,Y 168.858,Z 469.745,A -85,B 0,C 180,E1 -22933.157,E2 -22933.157} C_VEL
LIN {X 0,Y 169.687,Z 466.6,A -85,B 0,C 180,E1 -22936.835,E2 -22936.835} C_VEL
LIN {X 0,Y 170.948,Z 462.185,A -85,B 0,C 180,E1 -22940.578,E2 -22940.578} C_VEL
LIN {X 0,Y 172.626,Z 456.634,A -85,B 0,C 180,E1 -22944.16,E2 -22944.16} C_VEL
LIN {X 0,Y 174.911,Z 449.573,A -85,B 0,C 180,E1 -22947.699,E2 -22947.699} C_VEL
LIN {X 0,Y 177.217,Z 442.345,A -85,B 0,C 180,E1 -22950.57,E2 -22950.57} C_VEL
LIN {X 0,Y 179.936,Z 433.58,A -85,B 0,C 180,E1 -22953.361,E2 -22953.361} C_VEL
LIN {X 0,Y 183.054,Z 422.667,A -85,B 0,C 180,E1 -22956.062,E2 -22956.062} C_VEL
LIN {X 0,Y 185.866,Z 411.592,A -85,B 0,C 180,E1 -22958.193,E2 -22958.193} C_VEL
LIN {X 0,Y 188.338,Z 399.724,A -85,B 0,C 180,E1 -22959.94,E2 -22959.94} C_VEL
LIN {X 0,Y 190.393,Z 387.16,A -85,B 0,C 180,E1 -22961.311,E2 -22961.311} C_VEL
LIN {X 0,Y 192.009,Z 374.165,A -85,B 0,C 180,E1 -22962.285,E2 -22962.285} C_VEL
LIN {X 0,Y 193.151,Z 358.532,A -85,B 0,C 180,E1 -22962.959,E2 -22962.959} C_VEL
LIN {X 0,Y 195.336,Z 314.969,A -85,B 0,C 180,E1 -22964.527,E2 -22964.527} C_VEL
LIN {X 0,Y 189.914,Z 300.361,A -85,B 0,C 180,E1 -22966.265,E2 -22966.265} C_VEL
LIN {X 0,Y 183.326,Z 286.036,A -85,B 0,C 180,E1 -22968.362,E2 -22968.362} C_VEL
LIN {X 0,Y 176.16,Z 273.902,A -85,B 0,C 180,E1 -22970.705,E2 -22970.705} C_VEL
LIN {X 0,Y 173.372,Z 269.679,A -85,B 0,C 180,E1 -22971.657,E2 -22971.657} C_VEL
LIN {X 0,Y 171.698,Z 266.793,A -85,B 0,C 180,E1 -22972.326,E2 -22972.326} C_VEL
LIN {X 0,Y 171.449,Z 265.715,A -85,B 0,C 180,E1 -22972.919,E2 -22972.919} C_VEL
LIN {X 0,Y 171.365,Z 265.639,A -85,B 0,C 180,E1 -22976.818,E2 -22976.818} C_VEL
LIN {X 0,Y 171.394,Z 265.622,A -85,B 0,C 180,E1 -22980.578,E2 -22980.578} C_VEL
LIN {X 0,Y 171.371,Z 265.614,A -85,B 0,C 180,E1 -22985.042,E2 -22985.042} C_VEL
LIN {X 0,Y 171.331,Z 265.645,A -85,B 0,C 180,E1 -22988.811,E2 -22988.811} C_VEL
LIN {X 0,Y 171.3,Z 265.624,A -85,B 0,C 180,E1 -22994.226,E2 -22994.226} C_VEL
LIN {X 0,Y 171.315,Z 265.622,A -85,B 0,C 180,E1 -22998.988,E2 -22998.988} C_VEL
LIN {X 0,Y 171.346,Z 265.602,A -85,B 0,C 180,E1 -23002.042,E2 -23002.042} C_VEL
LIN {X 0,Y 171.385,Z 265.632,A -85,B 0,C 180,E1 -23005.101,E2 -23005.101} C_VEL
LIN {X 0,Y 171.382,Z 265.59,A -85,B 0,C 180,E1 -23010.532,E2 -23010.532} C_VEL
LIN {X 0,Y 171.398,Z 265.631,A -85,B 0,C 180,E1 -23015.802,E2 -23015.802} C_VEL
LIN {X 0,Y 171.507,Z 265.574,A -85,B 0,C 180,E1 -23020.872,E2 -23020.872} C_VEL
LIN {X 0,Y 171.558,Z 265.594,A -85,B 0,C 180,E1 -23025.78,E2 -23025.78} C_VEL
LIN {X 0,Y 171.843,Z 265.56,A -85,B 0,C 180,E1 -23030.593,E2 -23030.593} C_VEL
LIN {X 0,Y 171.782,Z 265.537,A -85,B 0,C 180,E1 -23035.315,E2 -23035.315} C_VEL
LIN {X 0,Y 172.313,Z 265.52,A -85,B 0,C 180,E1 -23040.008,E2 -23040.008} C_VEL
LIN {X 0,Y 171.868,Z 265.538,A -85,B 0,C 180,E1 -23047.054,E2 -23047.054} C_VEL
LIN {X 0,Y 171.777,Z 265.587,A -85,B 0,C 180,E1 -23050.903,E2 -23050.903} C_VEL
LIN {X 0,Y 171.534,Z 265.584,A -85,B 0,C 180,E1 -23056.674,E2 -23056.674} C_VEL
LIN {X 0,Y 171.527,Z 265.62,A -85,B 0,C 180,E1 -23059.54,E2 -23059.54} C_VEL
LIN {X 0,Y 171.457,Z 265.603,A -85,B 0,C 180,E1 -23065.604,E2 -23065.604} C_VEL
LIN {X 0,Y 171.432,Z 265.608,A -85,B 0,C 180,E1 -23070.578,E2 -23070.578} C_VEL
LIN {X 0,Y 171.407,Z 265.633,A -85,B 0,C 180,E1 -23075.04,E2 -23075.04} C_VEL
LIN {X 0,Y 171.359,Z 265.627,A -85,B 0,C 180,E1 -23078.805,E2 -23078.805} C_VEL
LIN {X 0,Y 171.363,Z 265.795,A -85,B 0,C 180,E1 -23083.959,E2 -23083.959} C_VEL
LIN {X 0,Y 171.605,Z 266.806,A -85,B 0,C 180,E1 -23084.486,E2 -23084.486} C_VEL
LIN {X 0,Y 173.307,Z 269.748,A -85,B 0,C 180,E1 -23085.159,E2 -23085.159} C_VEL
LIN {X 0,Y 178.921,Z 279.917,A -85,B 0,C 180,E1 -23087.131,E2 -23087.131} C_VEL
LIN {X 0,Y 185.874,Z 294.577,A -85,B 0,C 180,E1 -23089.452,E2 -23089.452} C_VEL
LIN {X 0,Y 193.109,Z 312.672,A -85,B 0,C 180,E1 -23091.777,E2 -23091.777} C_VEL
LIN {X 0,Y 194.662,Z 317.53,A -85,B 0,C 180,E1 -23092.294,E2 -23092.294} C_VEL
LIN {X 0,Y 195.222,Z 322.888,A -85,B 0,C 180,E1 -23092.641,E2 -23092.641} C_VEL
LIN {X 0,Y 192.306,Z 374.892,A -85,B 0,C 180,E1 -23094.536,E2 -23094.536} C_VEL
LIN {X 0,Y 190.759,Z 388.424,A -85,B 0,C 180,E1 -23095.415,E2 -23095.415} C_VEL
LIN {X 0,Y 188.673,Z 401.24,A -85,B 0,C 180,E1 -23096.67,E2 -23096.67} C_VEL
LIN {X 0,Y 186.038,Z 413.785,A -85,B 0,C 180,E1 -23098.387,E2 -23098.387} C_VEL
LIN {X 0,Y 185.73,Z 415.19,A -85,B 0,C 180,E1 -23098.609,E2 -23098.609} C_VEL
LIN {X 0,Y 183.944,Z 420.245,A -85,B 0,C 180,E1 -23099.379,E2 -23099.379} C_VEL
LIN {X 0,Y 179.202,Z 428.073,A -85,B 0,C 180,E1 -23100.592,E2 -23100.592} C_VEL
LIN {X 0,Y 174.337,Z 435.418,A -85,B 0,C 180,E1 -23102.071,E2 -23102.071} C_VEL
LIN {X 0,Y 172.399,Z 439.716,A -85,B 0,C 180,E1 -23103.246,E2 -23103.246} C_VEL
LIN {X 0,Y 169.735,Z 448.272,A -85,B 0,C 180,E1 -23106.188,E2 -23106.188} C_VEL
LIN {X 0,Y 167.019,Z 456.342,A -85,B 0,C 180,E1 -23109.685,E2 -23109.685} C_VEL
LIN {X 0,Y 165.104,Z 461.784,A -85,B 0,C 180,E1 -23112.662,E2 -23112.662} C_VEL
LIN {X 0,Y 163.514,Z 467.111,A -85,B 0,C 180,E1 -23116.324,E2 -23116.324} C_VEL
LIN {X 0,Y 162.463,Z 471.236,A -85,B 0,C 180,E1 -23120.034,E2 -23120.034} C_VEL
LIN {X 0,Y 162.036,Z 473.38,A -85,B 0,C 180,E1 -23122.522,E2 -23122.522} C_VEL
LIN {X 0,Y 161.787,Z 475.06,A -85,B 0,C 180,E1 -23125.014,E2 -23125.014} C_VEL
LIN {X 0,Y 161.709,Z 476.765,A -85,B 0,C 180,E1 -23128.628,E2 -23128.628} C_VEL
LIN {X 0,Y 161.742,Z 477.551,A -85,B 0,C 180,E1 -23131.804,E2 -23131.804} C_VEL
LIN {X 0,Y 161.788,Z 477.656,A -85,B 0,C 180,E1 -23134.982,E2 -23134.982} C_VEL
LIN {X 0,Y 162.56,Z 476.578,A -85,B 0,C 180,E1 -23139.956,E2 -23139.956} C_VEL
LIN {X 0,Y 163.27,Z 475.432,A -85,B 0,C 180,E1 -23142.427,E2 -23142.427} C_VEL
LIN {X 0,Y 164.267,Z 473.866,A -85,B 0,C 180,E1 -23144.872,E2 -23144.872} C_VEL
LIN {X 0,Y 166.197,Z 470.742,A -85,B 0,C 180,E1 -23148.489,E2 -23148.489} C_VEL
LIN {X 0,Y 168.923,Z 466.58,A -85,B 0,C 180,E1 -23151.988,E2 -23151.988} C_VEL
LIN {X 0,Y 172.687,Z 460.271,A -85,B 0,C 180,E1 -23155.942,E2 -23155.942} C_VEL
LIN {X 0,Y 176.528,Z 453.43,A -85,B 0,C 180,E1 -23159.187,E2 -23159.187} C_VEL
LIN {X 0,Y 180.968,Z 444.924,A -85,B 0,C 180,E1 -23162.273,E2 -23162.273} C_VEL
LIN {X 0,Y 185.176,Z 436.22,A -85,B 0,C 180,E1 -23164.699,E2 -23164.699} C_VEL
LIN {X 0,Y 189.65,Z 425.557,A -85,B 0,C 180,E1 -23167.024,E2 -23167.024} C_VEL
LIN {X 0,Y 193.476,Z 414.934,A -85,B 0,C 180,E1 -23168.797,E2 -23168.797} C_VEL
LIN {X 0,Y 196.984,Z 403.098,A -85,B 0,C 180,E1 -23170.288,E2 -23170.288} C_VEL
LIN {X 0,Y 199.774,Z 390.905,A -85,B 0,C 180,E1 -23171.436,E2 -23171.436} C_VEL
LIN {X 0,Y 202.03,Z 377.714,A -85,B 0,C 180,E1 -23172.263,E2 -23172.263} C_VEL
LIN {X 0,Y 203.45,Z 362.283,A -85,B 0,C 180,E1 -23172.865,E2 -23172.865} C_VEL
LIN {X 0,Y 205.661,Z 331.828,A -85,B 0,C 180,E1 -23173.861,E2 -23173.861} C_VEL
LIN {X 0,Y 201.524,Z 321.413,A -85,B 0,C 180,E1 -23175.943,E2 -23175.943} C_VEL
LIN {X 0,Y 197.445,Z 312.719,A -85,B 0,C 180,E1 -23178.1,E2 -23178.1} C_VEL
LIN {X 0,Y 192.569,Z 303.692,A -85,B 0,C 180,E1 -23180.927,E2 -23180.927} C_VEL
LIN {X 0,Y 189.441,Z 298.471,A -85,B 0,C 180,E1 -23182.918,E2 -23182.918} C_VEL
LIN {X 0,Y 186.617,Z 293.949,A -85,B 0,C 180,E1 -23184.921,E2 -23184.921} C_VEL
LIN {X 0,Y 183.471,Z 289.143,A -85,B 0,C 180,E1 -23187.401,E2 -23187.401} C_VEL
LIN {X 0,Y 180.438,Z 285.419,A -85,B 0,C 180,E1 -23190.099,E2 -23190.099} C_VEL
LIN {X 0,Y 179.483,Z 283.864,A -85,B 0,C 180,E1 -23191.095,E2 -23191.095} C_VEL
LIN {X 0,Y 176.984,Z 281.746,A -85,B 0,C 180,E1 -23193.815,E2 -23193.815} C_VEL
LIN {X 0,Y 175.281,Z 278.501,A -85,B 0,C 180,E1 -23196.354,E2 -23196.354} C_VEL
LIN {X 0,Y 172.45,Z 276.595,A -85,B 0,C 180,E1 -23201.581,E2 -23201.581} C_VEL
LIN {X 0,Y 171.242,Z 274.479,A -85,B 0,C 180,E1 -23208.151,E2 -23208.151} C_VEL
LIN {X 0,Y 171.429,Z 274.595,A -85,B 0,C 180,E1 -23211.149,E2 -23211.149} C_VEL
LIN {X 0,Y 175.763,Z 278.504,A -85,B 0,C 180,E1 -23221.51,E2 -23221.51} C_VEL
LIN {X 0,Y 177.05,Z 281.319,A -85,B 0,C 180,E1 -23223.441,E2 -23223.441} C_VEL
LIN {X 0,Y 179.536,Z 283.655,A -85,B 0,C 180,E1 -23226.172,E2 -23226.172} C_VEL
LIN {X 0,Y 180.296,Z 284.478,A -85,B 0,C 180,E1 -23226.919,E2 -23226.919} C_VEL
LIN {X 0,Y 182.798,Z 288.174,A -85,B 0,C 180,E1 -23229.277,E2 -23229.277} C_VEL
LIN {X 0,Y 184.06,Z 289.555,A -85,B 0,C 180,E1 -23230.289,E2 -23230.289} C_VEL
LIN {X 0,Y 186.959,Z 293.503,A -85,B 0,C 180,E1 -23232.491,E2 -23232.491} C_VEL
LIN {X 0,Y 191.069,Z 299.454,A -85,B 0,C 180,E1 -23235.254,E2 -23235.254} C_VEL
LIN {X 0,Y 193.882,Z 303.723,A -85,B 0,C 180,E1 -23236.946,E2 -23236.946} C_VEL
LIN {X 0,Y 198.502,Z 312.099,A -85,B 0,C 180,E1 -23239.539,E2 -23239.539} C_VEL
LIN {X 0,Y 203.842,Z 323.564,A -85,B 0,C 180,E1 -23242.279,E2 -23242.279} C_VEL
LIN {X 0,Y 205.838,Z 328.472,A -85,B 0,C 180,E1 -23243.253,E2 -23243.253} C_VEL
LIN {X 0,Y 202.55,Z 371.149,A -85,B 0,C 180,E1 -23244.696,E2 -23244.696} C_VEL
LIN {X 0,Y 200.619,Z 383.957,A -85,B 0,C 180,E1 -23245.429,E2 -23245.429} C_VEL
LIN {X 0,Y 198.191,Z 395.745,A -85,B 0,C 180,E1 -23246.447,E2 -23246.447} C_VEL
LIN {X 0,Y 195.037,Z 407.611,A -85,B 0,C 180,E1 -23247.865,E2 -23247.865} C_VEL
LIN {X 0,Y 191.124,Z 419.237,A -85,B 0,C 180,E1 -23249.692,E2 -23249.692} C_VEL
LIN {X 0,Y 187.216,Z 429.08,A -85,B 0,C 180,E1 -23251.696,E2 -23251.696} C_VEL
LIN {X 0,Y 182.759,Z 438.791,A -85,B 0,C 180,E1 -23254.234,E2 -23254.234} C_VEL
LIN {X 0,Y 178.42,Z 447.215,A -85,B 0,C 180,E1 -23257.102,E2 -23257.102} C_VEL
LIN {X 0,Y 174.574,Z 454.083,A -85,B 0,C 180,E1 -23260.105,E2 -23260.105} C_VEL
LIN {X 0,Y 170.771,Z 460.476,A -85,B 0,C 180,E1 -23263.746,E2 -23263.746} C_VEL
LIN {X 0,Y 167.406,Z 465.7,A -85,B 0,C 180,E1 -23267.804,E2 -23267.804} C_VEL
LIN {X 0,Y 164.897,Z 469.349,A -85,B 0,C 180,E1 -23271.833,E2 -23271.833} C_VEL
LIN {X 0,Y 163.141,Z 471.772,A -85,B 0,C 180,E1 -23275.945,E2 -23275.945} C_VEL
LIN {X 0,Y 161.944,Z 473.071,A -85,B 0,C 180,E1 -23280.201,E2 -23280.201} C_VEL
LIN {X 0,Y 161.311,Z 473.23,A -85,B 0,C 180,E1 -23284.174,E2 -23284.174} C_VEL
LIN {X 0,Y 161.243,Z 472.782,A -85,B 0,C 180,E1 -23286.906,E2 -23286.906} C_VEL
LIN {X 0,Y 161.284,Z 471.829,A -85,B 0,C 180,E1 -23289.601,E2 -23289.601} C_VEL
LIN {X 0,Y 161.705,Z 470.03,A -85,B 0,C 180,E1 -23292.936,E2 -23292.936} C_VEL
LIN {X 0,Y 162.412,Z 467.441,A -85,B 0,C 180,E1 -23296.234,E2 -23296.234} C_VEL
LIN {X 0,Y 163.814,Z 462.737,A -85,B 0,C 180,E1 -23300.599,E2 -23300.599} C_VEL
LIN {X 0,Y 165.619,Z 456.978,A -85,B 0,C 180,E1 -23304.523,E2 -23304.523} C_VEL
LIN {X 0,Y 168.211,Z 449.335,A -85,B 0,C 180,E1 -23308.502,E2 -23308.502} C_VEL
LIN {X 0,Y 170.922,Z 441.209,A -85,B 0,C 180,E1 -23311.769,E2 -23311.769} C_VEL
LIN {X 0,Y 174.138,Z 431.109,A -85,B 0,C 180,E1 -23314.922,E2 -23314.922} C_VEL
LIN {X 0,Y 177.17,Z 420.673,A -85,B 0,C 180,E1 -23317.461,E2 -23317.461} C_VEL
LIN {X 0,Y 180.028,Z 409.48,A -85,B 0,C 180,E1 -23319.552,E2 -23319.552} C_VEL
LIN {X 0,Y 182.671,Z 396.71,A -85,B 0,C 180,E1 -23321.374,E2 -23321.374} C_VEL
LIN {X 0,Y 184.666,Z 384.363,A -85,B 0,C 180,E1 -23322.642,E2 -23322.642} C_VEL
LIN {X 0,Y 186.294,Z 370.237,A -85,B 0,C 180,E1 -23323.597,E2 -23323.597} C_VEL
LIN {X 0,Y 189.42,Z 317.269,A -85,B 0,C 180,E1 -23325.564,E2 -23325.564} C_VEL
LIN {X 0,Y 184.712,Z 304.212,A -85,B 0,C 180,E1 -23327.156,E2 -23327.156} C_VEL
LIN {X 0,Y 178.28,Z 289.999,A -85,B 0,C 180,E1 -23329.329,E2 -23329.329} C_VEL
LIN {X 0,Y 171.574,Z 278.603,A -85,B 0,C 180,E1 -23331.635,E2 -23331.635} C_VEL
LIN {X 0,Y 166.445,Z 270.732,A -85,B 0,C 180,E1 -23333.506,E2 -23333.506} C_VEL
LIN {X 0,Y 164.742,Z 268.042,A -85,B 0,C 180,E1 -23334.194,E2 -23334.194} C_VEL
LIN {X 0,Y 164.438,Z 266.896,A -85,B 0,C 180,E1 -23334.629,E2 -23334.629} C_VEL
LIN {X 0,Y 164.37,Z 266.516,A -85,B 0,C 180,E1 -23335.316,E2 -23335.316} C_VEL
LIN {X 0,Y 164.334,Z 266.507,A -85,B 0,C 180,E1 -23341.223,E2 -23341.223} C_VEL
LIN {X 0,Y 164.271,Z 266.505,A -85,B 0,C 180,E1 -23346.798,E2 -23346.798} C_VEL
LIN {X 0,Y 164.268,Z 266.514,A -85,B 0,C 180,E1 -23349.925,E2 -23349.925} C_VEL
LIN {X 0,Y 164.263,Z 266.494,A -85,B 0,C 180,E1 -23353.35,E2 -23353.35} C_VEL
LIN {X 0,Y 164.245,Z 266.527,A -85,B 0,C 180,E1 -23356.806,E2 -23356.806} C_VEL
LIN {X 0,Y 164.274,Z 266.484,A -85,B 0,C 180,E1 -23360.363,E2 -23360.363} C_VEL
LIN {X 0,Y 164.313,Z 266.503,A -85,B 0,C 180,E1 -23364.36,E2 -23364.36} C_VEL
LIN {X 0,Y 164.346,Z 266.478,A -85,B 0,C 180,E1 -23369.136,E2 -23369.136} C_VEL
LIN {X 0,Y 164.349,Z 266.496,A -85,B 0,C 180,E1 -23374.693,E2 -23374.693} C_VEL
LIN {X 0,Y 164.413,Z 266.466,A -85,B 0,C 180,E1 -23380.126,E2 -23380.126} C_VEL
LIN {X 0,Y 164.485,Z 266.462,A -85,B 0,C 180,E1 -23385.155,E2 -23385.155} C_VEL
LIN {X 0,Y 164.764,Z 266.447,A -85,B 0,C 180,E1 -23390.185,E2 -23390.185} C_VEL
LIN {X 0,Y 164.82,Z 266.404,A -85,B 0,C 180,E1 -23392.659,E2 -23392.659} C_VEL
LIN {X 0,Y 165.277,Z 266.396,A -85,B 0,C 180,E1 -23400.008,E2 -23400.008} C_VEL
LIN {X 0,Y 164.83,Z 266.417,A -85,B 0,C 180,E1 -23407.357,E2 -23407.357} C_VEL
LIN {X 0,Y 164.712,Z 266.467,A -85,B 0,C 180,E1 -23411.067,E2 -23411.067} C_VEL
LIN {X 0,Y 164.463,Z 266.472,A -85,B 0,C 180,E1 -23417.413,E2 -23417.413} C_VEL
LIN {X 0,Y 164.461,Z 266.5,A -85,B 0,C 180,E1 -23419.999,E2 -23419.999} C_VEL
LIN {X 0,Y 164.384,Z 266.489,A -85,B 0,C 180,E1 -23426.123,E2 -23426.123} C_VEL
LIN {X 0,Y 164.367,Z 266.486,A -85,B 0,C 180,E1 -23431.22,E2 -23431.22} C_VEL
LIN {X 0,Y 164.295,Z 266.502,A -85,B 0,C 180,E1 -23436.798,E2 -23436.798} C_VEL
LIN {X 0,Y 164.325,Z 266.725,A -85,B 0,C 180,E1 -23442.046,E2 -23442.046} C_VEL
LIN {X 0,Y 164.604,Z 267.826,A -85,B 0,C 180,E1 -23442.578,E2 -23442.578} C_VEL
LIN {X 0,Y 166.147,Z 270.505,A -85,B 0,C 180,E1 -23443.224,E2 -23443.224} C_VEL
LIN {X 0,Y 167.208,Z 271.883,A -85,B 0,C 180,E1 -23443.612,E2 -23443.612} C_VEL
LIN {X 0,Y 170.301,Z 277.157,A -85,B 0,C 180,E1 -23444.773,E2 -23444.773} C_VEL
LIN {X 0,Y 175.922,Z 287.923,A -85,B 0,C 180,E1 -23446.819,E2 -23446.819} C_VEL
LIN {X 0,Y 182.308,Z 302.151,A -85,B 0,C 180,E1 -23449.052,E2 -23449.052} C_VEL
LIN {X 0,Y 188.625,Z 318.83,A -85,B 0,C 180,E1 -23451.182,E2 -23451.182} C_VEL
LIN {X 0,Y 189.225,Z 323.346,A -85,B 0,C 180,E1 -23451.516,E2 -23451.516} C_VEL
LIN {X 0,Y 186.339,Z 373.771,A -85,B 0,C 180,E1 -23453.386,E2 -23453.386} C_VEL
LIN {X 0,Y 184.69,Z 387.613,A -85,B 0,C 180,E1 -23454.275,E2 -23454.275} C_VEL
LIN {X 0,Y 182.513,Z 400.663,A -85,B 0,C 180,E1 -23455.556,E2 -23455.556} C_VEL
LIN {X 0,Y 179.977,Z 412.519,A -85,B 0,C 180,E1 -23457.191,E2 -23457.191} C_VEL
LIN {X 0,Y 177.032,Z 423.944,A -85,B 0,C 180,E1 -23459.259,E2 -23459.259} C_VEL
LIN {X 0,Y 174.067,Z 434.256,A -85,B 0,C 180,E1 -23461.677,E2 -23461.677} C_VEL
LIN {X 0,Y 172.399,Z 439.716,A -85,B 0,C 180,E1 -23463.246,E2 -23463.246} C_VEL
LIN {X 0,Y 170.5,Z 443.879,A -85,B 0,C 180,E1 -23464.513,E2 -23464.513} C_VEL
LIN {X 0,Y 165.721,Z 450.162,A -85,B 0,C 180,E1 -23466.571,E2 -23466.571} C_VEL
LIN {X 0,Y 160.964,Z 455.827,A -85,B 0,C 180,E1 -23468.894,E2 -23468.894} C_VEL
LIN {X 0,Y 159.15,Z 459.019,A -85,B 0,C 180,E1 -23470.541,E2 -23470.541} C_VEL
LIN {X 0,Y 157.056,Z 465.052,A -85,B 0,C 180,E1 -23474.423,E2 -23474.423} C_VEL
LIN {X 0,Y 155.79,Z 469.637,A -85,B 0,C 180,E1 -23478.285,E2 -23478.285} C_VEL
LIN {X 0,Y 154.984,Z 473.101,A -85,B 0,C 180,E1 -23482.179,E2 -23482.179} C_VEL
LIN {X 0,Y 154.717,Z 474.818,A -85,B 0,C 180,E1 -23484.785,E2 -23484.785} C_VEL
LIN {X 0,Y 154.652,Z 476.765,A -85,B 0,C 180,E1 -23489.148,E2 -23489.148} C_VEL
LIN {X 0,Y 154.649,Z 477.511,A -85,B 0,C 180,E1 -23492.603,E2 -23492.603} C_VEL
LIN {X 0,Y 155.012,Z 477.256,A -85,B 0,C 180,E1 -23497.815,E2 -23497.815} C_VEL
LIN {X 0,Y 156.331,Z 475.473,A -85,B 0,C 180,E1 -23502.988,E2 -23502.988} C_VEL
LIN {X 0,Y 157.386,Z 473.945,A -85,B 0,C 180,E1 -23505.539,E2 -23505.539} C_VEL
LIN {X 0,Y 159.462,Z 470.891,A -85,B 0,C 180,E1 -23509.3,E2 -23509.3} C_VEL
LIN {X 0,Y 162.371,Z 466.81,A -85,B 0,C 180,E1 -23512.924,E2 -23512.924} C_VEL
LIN {X 0,Y 166.337,Z 460.601,A -85,B 0,C 180,E1 -23517.011,E2 -23517.011} C_VEL
LIN {X 0,Y 170.374,Z 453.87,A -85,B 0,C 180,E1 -23520.35,E2 -23520.35} C_VEL
LIN {X 0,Y 175.041,Z 445.532,A -85,B 0,C 180,E1 -23523.506,E2 -23523.506} C_VEL
LIN {X 0,Y 179.422,Z 436.967,A -85,B 0,C 180,E1 -23525.981,E2 -23525.981} C_VEL
LIN {X 0,Y 184.077,Z 426.472,A -85,B 0,C 180,E1 -23528.344,E2 -23528.344} C_VEL
LIN {X 0,Y 188.055,Z 416.096,A -85,B 0,C 180,E1 -23530.138,E2 -23530.138} C_VEL
LIN {X 0,Y 191.688,Z 404.697,A -85,B 0,C 180,E1 -23531.644,E2 -23531.644} C_VEL
LIN {X 0,Y 194.854,Z 391.777,A -85,B 0,C 180,E1 -23532.902,E2 -23532.902} C_VEL
LIN {X 0,Y 197.283,Z 378.57,A -85,B 0,C 180,E1 -23533.762,E2 -23533.762} C_VEL
LIN {X 0,Y 198.7,Z 364.696,A -85,B 0,C 180,E1 -23534.336,E2 -23534.336} C_VEL
LIN {X 0,Y 200.999,Z 334.245,A -85,B 0,C 180,E1 -23535.351,E2 -23535.351} C_VEL
LIN {X 0,Y 197.063,Z 324.174,A -85,B 0,C 180,E1 -23537.502,E2 -23537.502} C_VEL
LIN {X 0,Y 193.264,Z 316.136,A -85,B 0,C 180,E1 -23539.686,E2 -23539.686} C_VEL
LIN {X 0,Y 189.048,Z 308.167,A -85,B 0,C 180,E1 -23542.349,E2 -23542.349} C_VEL
LIN {X 0,Y 186.58,Z 303.849,A -85,B 0,C 180,E1 -23544.069,E2 -23544.069} C_VEL
LIN {X 0,Y 184.175,Z 299.866,A -85,B 0,C 180,E1 -23545.897,E2 -23545.897} C_VEL
LIN {X 0,Y 181.454,Z 295.494,A -85,B 0,C 180,E1 -23548.184,E2 -23548.184} C_VEL
LIN {X 0,Y 178.622,Z 291.842,A -85,B 0,C 180,E1 -23550.876,E2 -23550.876} C_VEL
LIN {X 0,Y 177.739,Z 290.547,A -85,B 0,C 180,E1 -23551.827,E2 -23551.827} C_VEL
LIN {X 0,Y 175.319,Z 288.144,A -85,B 0,C 180,E1 -23554.678,E2 -23554.678} C_VEL
LIN {X 0,Y 173.899,Z 285.354,A -85,B 0,C 180,E1 -23556.947,E2 -23556.947} C_VEL
LIN {X 0,Y 170.311,Z 281.559,A -85,B 0,C 180,E1 -23568.085,E2 -23568.085} C_VEL
LIN {X 0,Y 170.485,Z 281.652,A -85,B 0,C 180,E1 -23571.099,E2 -23571.099} C_VEL
LIN {X 0,Y 174.357,Z 285.38,A -85,B 0,C 180,E1 -23580.922,E2 -23580.922} C_VEL
LIN {X 0,Y 175.748,Z 288.244,A -85,B 0,C 180,E1 -23583.072,E2 -23583.072} C_VEL
LIN {X 0,Y 178.542,Z 291.059,A -85,B 0,C 180,E1 -23586.206,E2 -23586.206} C_VEL
LIN {X 0,Y 181.125,Z 294.864,A -85,B 0,C 180,E1 -23588.745,E2 -23588.745} C_VEL
LIN {X 0,Y 182.248,Z 296.339,A -85,B 0,C 180,E1 -23589.726,E2 -23589.726} C_VEL
LIN {X 0,Y 185.667,Z 301.201,A -85,B 0,C 180,E1 -23592.4,E2 -23592.4} C_VEL
LIN {X 0,Y 189.019,Z 306.246,A -85,B 0,C 180,E1 -23594.731,E2 -23594.731} C_VEL
LIN {X 0,Y 191.397,Z 310.039,A -85,B 0,C 180,E1 -23596.226,E2 -23596.226} C_VEL
LIN {X 0,Y 195.408,Z 317.773,A -85,B 0,C 180,E1 -23598.632,E2 -23598.632} C_VEL
LIN {X 0,Y 200.057,Z 328.079,A -85,B 0,C 180,E1 -23601.165,E2 -23601.165} C_VEL
LIN {X 0,Y 201.208,Z 331.043,A -85,B 0,C 180,E1 -23601.777,E2 -23601.777} C_VEL
LIN {X 0,Y 197.99,Z 370.967,A -85,B 0,C 180,E1 -23603.14,E2 -23603.14} C_VEL
LIN {X 0,Y 196.133,Z 383.06,A -85,B 0,C 180,E1 -23603.82,E2 -23603.82} C_VEL
LIN {X 0,Y 193.571,Z 395.007,A -85,B 0,C 180,E1 -23604.819,E2 -23604.819} C_VEL
LIN {X 0,Y 190.155,Z 407.567,A -85,B 0,C 180,E1 -23606.319,E2 -23606.319} C_VEL
LIN {X 0,Y 186.201,Z 418.84,A -85,B 0,C 180,E1 -23608.087,E2 -23608.087} C_VEL
LIN {X 0,Y 182.145,Z 428.7,A -85,B 0,C 180,E1 -23610.096,E2 -23610.096} C_VEL
LIN {X 0,Y 177.414,Z 438.571,A -85,B 0,C 180,E1 -23612.675,E2 -23612.675} C_VEL
LIN {X 0,Y 172.83,Z 447.041,A -85,B 0,C 180,E1 -23615.586,E2 -23615.586} C_VEL
LIN {X 0,Y 168.717,Z 453.969,A -85,B 0,C 180,E1 -23618.658,E2 -23618.658} C_VEL
LIN {X 0,Y 165.17,Z 459.59,A -85,B 0,C 180,E1 -23621.877,E2 -23621.877} C_VEL
LIN {X 0,Y 161.544,Z 464.902,A -85,B 0,C 180,E1 -23625.89,E2 -23625.89} C_VEL
LIN {X 0,Y 158.678,Z 468.835,A -85,B 0,C 180,E1 -23630.046,E2 -23630.046} C_VEL
LIN {X 0,Y 156.596,Z 471.499,A -85,B 0,C 180,E1 -23634.31,E2 -23634.31} C_VEL
LIN {X 0,Y 154.971,Z 473.147,A -85,B 0,C 180,E1 -23639.482,E2 -23639.482} C_VEL
LIN {X 0,Y 154.356,Z 473.389,A -85,B 0,C 180,E1 -23642.918,E2 -23642.918} C_VEL
LIN {X 0,Y 154.144,Z 473.05,A -85,B 0,C 180,E1 -23645.776,E2 -23645.776} C_VEL
LIN {X 0,Y 154.128,Z 472.276,A -85,B 0,C 180,E1 -23648.608,E2 -23648.608} C_VEL
LIN {X 0,Y 154.552,Z 470.277,A -85,B 0,C 180,E1 -23652.699,E2 -23652.699} C_VEL
LIN {X 0,Y 155.469,Z 467.078,A -85,B 0,C 180,E1 -23656.939,E2 -23656.939} C_VEL
LIN {X 0,Y 156.997,Z 462.168,A -85,B 0,C 180,E1 -23661.477,E2 -23661.477} C_VEL
LIN {X 0,Y 158.961,Z 456.234,A -85,B 0,C 180,E1 -23665.565,E2 -23665.565} C_VEL
LIN {X 0,Y 161.621,Z 448.807,A -85,B 0,C 180,E1 -23669.484,E2 -23669.484} C_VEL
LIN {X 0,Y 164.706,Z 439.945,A -85,B 0,C 180,E1 -23673.059,E2 -23673.059} C_VEL
LIN {X 0,Y 167.787,Z 430.596,A -85,B 0,C 180,E1 -23676.013,E2 -23676.013} C_VEL
LIN {X 0,Y 170.736,Z 420.805,A -85,B 0,C 180,E1 -23678.449,E2 -23678.449} C_VEL
LIN {X 0,Y 173.58,Z 410.214,A -85,B 0,C 180,E1 -23680.5,E2 -23680.5} C_VEL
LIN {X 0,Y 176.315,Z 397.606,A -85,B 0,C 180,E1 -23682.373,E2 -23682.373} C_VEL
LIN {X 0,Y 178.389,Z 385.626,A -85,B 0,C 180,E1 -23683.675,E2 -23683.675} C_VEL
LIN {X 0,Y 180.058,Z 372.171,A -85,B 0,C 180,E1 -23684.653,E2 -23684.653} C_VEL
LIN {X 0,Y 181.453,Z 352.888,A -85,B 0,C 180,E1 -23685.446,E2 -23685.446} C_VEL
LIN {X 0,Y 183.407,Z 318.807,A -85,B 0,C 180,E1 -23686.715,E2 -23686.715} C_VEL
LIN {X 0,Y 178.711,Z 305.974,A -85,B 0,C 180,E1 -23688.399,E2 -23688.399} C_VEL
LIN {X 0,Y 172.839,Z 293.14,A -85,B 0,C 180,E1 -23690.506,E2 -23690.506} C_VEL
LIN {X 0,Y 166.83,Z 282.956,A -85,B 0,C 180,E1 -23692.682,E2 -23692.682} C_VEL
LIN {X 0,Y 161.999,Z 275.499,A -85,B 0,C 180,E1 -23694.553,E2 -23694.553} C_VEL
LIN {X 0,Y 159.635,Z 271.779,A -85,B 0,C 180,E1 -23695.536,E2 -23695.536} C_VEL
LIN {X 0,Y 157.854,Z 269.372,A -85,B 0,C 180,E1 -23696.28,E2 -23696.28} C_VEL
LIN {X 0,Y 157.359,Z 267.973,A -85,B 0,C 180,E1 -23696.739,E2 -23696.739} C_VEL
LIN {X 0,Y 157.261,Z 267.465,A -85,B 0,C 180,E1 -23697.192,E2 -23697.192} C_VEL
LIN {X 0,Y 157.246,Z 267.397,A -85,B 0,C 180,E1 -23702.437,E2 -23702.437} C_VEL
LIN {X 0,Y 157.245,Z 267.377,A -85,B 0,C 180,E1 -23706.455,E2 -23706.455} C_VEL
LIN {X 0,Y 157.171,Z 267.375,A -85,B 0,C 180,E1 -23712.126,E2 -23712.126} C_VEL
LIN {X 0,Y 157.174,Z 267.398,A -85,B 0,C 180,E1 -23717.891,E2 -23717.891} C_VEL
LIN {X 0,Y 157.245,Z 267.371,A -85,B 0,C 180,E1 -23723.565,E2 -23723.565} C_VEL
LIN {X 0,Y 157.264,Z 267.376,A -85,B 0,C 180,E1 -23728.117,E2 -23728.117} C_VEL
LIN {X 0,Y 157.258,Z 267.359,A -85,B 0,C 180,E1 -23733.465,E2 -23733.465} C_VEL
LIN {X 0,Y 157.355,Z 267.35,A -85,B 0,C 180,E1 -23739.711,E2 -23739.711} C_VEL
LIN {X 0,Y 157.416,Z 267.331,A -85,B 0,C 180,E1 -23744.472,E2 -23744.472} C_VEL
LIN {X 0,Y 157.687,Z 267.334,A -85,B 0,C 180,E1 -23749.74,E2 -23749.74} C_VEL
LIN {X 0,Y 157.759,Z 267.286,A -85,B 0,C 180,E1 -23752.329,E2 -23752.329} C_VEL
LIN {X 0,Y 158.24,Z 267.272,A -85,B 0,C 180,E1 -23760.009,E2 -23760.009} C_VEL
LIN {X 0,Y 157.768,Z 267.3,A -85,B 0,C 180,E1 -23767.688,E2 -23767.688} C_VEL
LIN {X 0,Y 157.642,Z 267.347,A -85,B 0,C 180,E1 -23771.236,E2 -23771.236} C_VEL
LIN {X 0,Y 157.433,Z 267.333,A -85,B 0,C 180,E1 -23775.545,E2 -23775.545} C_VEL
LIN {X 0,Y 157.369,Z 267.377,A -85,B 0,C 180,E1 -23780.942,E2 -23780.942} C_VEL
LIN {X 0,Y 157.324,Z 267.375,A -85,B 0,C 180,E1 -23786.687,E2 -23786.687} C_VEL
LIN {X 0,Y 157.279,Z 267.372,A -85,B 0,C 180,E1 -23792.436,E2 -23792.436} C_VEL
LIN {X 0,Y 157.274,Z 267.378,A -85,B 0,C 180,E1 -23796.449,E2 -23796.449} C_VEL
LIN {X 0,Y 157.276,Z 267.516,A -85,B 0,C 180,E1 -23799.728,E2 -23799.728} C_VEL
LIN {X 0,Y 157.537,Z 268.665,A -85,B 0,C 180,E1 -23800.358,E2 -23800.358} C_VEL
LIN {X 0,Y 159.071,Z 271.351,A -85,B 0,C 180,E1 -23801.083,E2 -23801.083} C_VEL
LIN {X 0,Y 160.117,Z 272.476,A -85,B 0,C 180,E1 -23801.495,E2 -23801.495} C_VEL
LIN {X 0,Y 162.225,Z 275.9,A -85,B 0,C 180,E1 -23802.371,E2 -23802.371} C_VEL
LIN {X 0,Y 165.733,Z 281.73,A -85,B 0,C 180,E1 -23803.765,E2 -23803.765} C_VEL
LIN {X 0,Y 171.613,Z 293.269,A -85,B 0,C 180,E1 -23806.018,E2 -23806.018} C_VEL
LIN {X 0,Y 177.641,Z 307.252,A -85,B 0,C 180,E1 -23808.251,E2 -23808.251} C_VEL
LIN {X 0,Y 183.023,Z 321.837,A -85,B 0,C 180,E1 -23810.183,E2 -23810.183} C_VEL
LIN {X 0,Y 183.146,Z 325.713,A -85,B 0,C 180,E1 -23810.4,E2 -23810.4} C_VEL
LIN {X 0,Y 180.189,Z 374.589,A -85,B 0,C 180,E1 -23812.273,E2 -23812.273} C_VEL
LIN {X 0,Y 178.518,Z 388.143,A -85,B 0,C 180,E1 -23813.19,E2 -23813.19} C_VEL
LIN {X 0,Y 176.245,Z 400.979,A -85,B 0,C 180,E1 -23814.498,E2 -23814.498} C_VEL
LIN {X 0,Y 173.624,Z 412.748,A -85,B 0,C 180,E1 -23816.179,E2 -23816.179} C_VEL
LIN {X 0,Y 170.568,Z 424.114,A -85,B 0,C 180,E1 -23818.307,E2 -23818.307} C_VEL
LIN {X 0,Y 167.486,Z 434.367,A -85,B 0,C 180,E1 -23820.802,E2 -23820.802} C_VEL
LIN {X 0,Y 164.217,Z 444.488,A -85,B 0,C 180,E1 -23824.008,E2 -23824.008} C_VEL
LIN {X 0,Y 161.7,Z 451.889,A -85,B 0,C 180,E1 -23826.971,E2 -23826.971} C_VEL
LIN {X 0,Y 159.15,Z 459.019,A -85,B 0,C 180,E1 -23830.541,E2 -23830.541} C_VEL
LIN {X 0,Y 157.443,Z 462.048,A -85,B 0,C 180,E1 -23832.273,E2 -23832.273} C_VEL
LIN {X 0,Y 153.218,Z 466.365,A -85,B 0,C 180,E1 -23835.177,E2 -23835.177} C_VEL
LIN {X 0,Y 149.314,Z 469.923,A -85,B 0,C 180,E1 -23838.368,E2 -23838.368} C_VEL
LIN {X 0,Y 148.16,Z 471.765,A -85,B 0,C 180,E1 -23840.493,E2 -23840.493} C_VEL
LIN {X 0,Y 147.645,Z 474.572,A -85,B 0,C 180,E1 -23844.535,E2 -23844.535} C_VEL
LIN {X 0,Y 147.546,Z 475.909,A -85,B 0,C 180,E1 -23847.268,E2 -23847.268} C_VEL
LIN {X 0,Y 147.607,Z 476.845,A -85,B 0,C 180,E1 -23849.998,E2 -23849.998} C_VEL
LIN {X 0,Y 147.547,Z 477.382,A -85,B 0,C 180,E1 -23852.728,E2 -23852.728} C_VEL
LIN {X 0,Y 147.647,Z 477.491,A -85,B 0,C 180,E1 -23855.461,E2 -23855.461} C_VEL
LIN {X 0,Y 148.561,Z 476.541,A -85,B 0,C 180,E1 -23860.905,E2 -23860.905} C_VEL
LIN {X 0,Y 149.414,Z 475.498,A -85,B 0,C 180,E1 -23863.6,E2 -23863.6} C_VEL
LIN {X 0,Y 150.537,Z 474.036,A -85,B 0,C 180,E1 -23866.265,E2 -23866.265} C_VEL
LIN {X 0,Y 152.771,Z 471.061,A -85,B 0,C 180,E1 -23870.181,E2 -23870.181} C_VEL
LIN {X 0,Y 155.868,Z 467.058,A -85,B 0,C 180,E1 -23873.939,E2 -23873.939} C_VEL
LIN {X 0,Y 160.055,Z 460.944,A -85,B 0,C 180,E1 -23878.164,E2 -23878.164} C_VEL
LIN {X 0,Y 164.312,Z 454.309,A -85,B 0,C 180,E1 -23881.596,E2 -23881.596} C_VEL
LIN {X 0,Y 169.204,Z 446.103,A -85,B 0,C 180,E1 -23884.825,E2 -23884.825} C_VEL
LIN {X 0,Y 173.764,Z 437.725,A -85,B 0,C 180,E1 -23887.347,E2 -23887.347} C_VEL
LIN {X 0,Y 178.605,Z 427.44,A -85,B 0,C 180,E1 -23889.746,E2 -23889.746} C_VEL
LIN {X 0,Y 183.287,Z 415.911,A -85,B 0,C 180,E1 -23891.774,E2 -23891.774} C_VEL
LIN {X 0,Y 187.063,Z 404.517,A -85,B 0,C 180,E1 -23893.284,E2 -23893.284} C_VEL
LIN {X 0,Y 190.35,Z 391.589,A -85,B 0,C 180,E1 -23894.545,E2 -23894.545} C_VEL
LIN {X 0,Y 192.892,Z 378.287,A -85,B 0,C 180,E1 -23895.399,E2 -23895.399} C_VEL
LIN {X 0,Y 194.424,Z 363.628,A -85,B 0,C 180,E1 -23895.993,E2 -23895.993} C_VEL
LIN {X 0,Y 196.503,Z 336.692,A -85,B 0,C 180,E1 -23896.911,E2 -23896.911} C_VEL
LIN {X 0,Y 192.707,Z 327.004,A -85,B 0,C 180,E1 -23899.163,E2 -23899.163} C_VEL
LIN {X 0,Y 188.913,Z 318.753,A -85,B 0,C 180,E1 -23901.586,E2 -23901.586} C_VEL
LIN {X 0,Y 184.425,Z 310.247,A -85,B 0,C 180,E1 -23904.786,E2 -23904.786} C_VEL
LIN {X 0,Y 181.392,Z 305.095,A -85,B 0,C 180,E1 -23907.237,E2 -23907.237} C_VEL
LIN {X 0,Y 179.442,Z 301.816,A -85,B 0,C 180,E1 -23909.031,E2 -23909.031} C_VEL
LIN {X 0,Y 176.753,Z 298.134,A -85,B 0,C 180,E1 -23911.756,E2 -23911.756} C_VEL
LIN {X 0,Y 176.116,Z 297.241,A -85,B 0,C 180,E1 -23912.474,E2 -23912.474} C_VEL
LIN {X 0,Y 173.808,Z 294.721,A -85,B 0,C 180,E1 -23915.401,E2 -23915.401} C_VEL
LIN {X 0,Y 172.702,Z 292.376,A -85,B 0,C 180,E1 -23917.279,E2 -23917.279} C_VEL
LIN {X 0,Y 169.381,Z 288.629,A -85,B 0,C 180,E1 -23928.019,E2 -23928.019} C_VEL
LIN {X 0,Y 169.563,Z 288.76,A -85,B 0,C 180,E1 -23931.214,E2 -23931.214} C_VEL
LIN {X 0,Y 172.944,Z 292.17,A -85,B 0,C 180,E1 -23940.272,E2 -23940.272} C_VEL
LIN {X 0,Y 174.517,Z 295.257,A -85,B 0,C 180,E1 -23942.773,E2 -23942.773} C_VEL
LIN {X 0,Y 176.813,Z 297.617,A -85,B 0,C 180,E1 -23945.481,E2 -23945.481} C_VEL
LIN {X 0,Y 179.377,Z 301.454,A -85,B 0,C 180,E1 -23948.122,E2 -23948.122} C_VEL
LIN {X 0,Y 183.362,Z 307.325,A -85,B 0,C 180,E1 -23951.53,E2 -23951.53} C_VEL
LIN {X 0,Y 187.618,Z 313.885,A -85,B 0,C 180,E1 -23954.606,E2 -23954.606} C_VEL
LIN {X 0,Y 191.996,Z 322.455,A -85,B 0,C 180,E1 -23957.429,E2 -23957.429} C_VEL
LIN {X 0,Y 196.429,Z 332.893,A -85,B 0,C 180,E1 -23960.061,E2 -23960.061} C_VEL
LIN {X 0,Y 196.712,Z 333.655,A -85,B 0,C 180,E1 -23960.223,E2 -23960.223} C_VEL
LIN {X 0,Y 193.547,Z 371.326,A -85,B 0,C 180,E1 -23961.527,E2 -23961.527} C_VEL
LIN {X 0,Y 191.505,Z 383.92,A -85,B 0,C 180,E1 -23962.245,E2 -23962.245} C_VEL
LIN {X 0,Y 188.836,Z 395.746,A -85,B 0,C 180,E1 -23963.255,E2 -23963.255} C_VEL
LIN {X 0,Y 185.564,Z 407.267,A -85,B 0,C 180,E1 -23964.642,E2 -23964.642} C_VEL
LIN {X 0,Y 181.445,Z 418.542,A -85,B 0,C 180,E1 -23966.405,E2 -23966.405} C_VEL
LIN {X 0,Y 177.185,Z 428.418,A -85,B 0,C 180,E1 -23968.413,E2 -23968.413} C_VEL
LIN {X 0,Y 172.219,Z 438.36,A -85,B 0,C 180,E1 -23971.026,E2 -23971.026} C_VEL
LIN {X 0,Y 167.385,Z 446.881,A -85,B 0,C 180,E1 -23973.983,E2 -23973.983} C_VEL
LIN {X 0,Y 162.201,Z 455.091,A -85,B 0,C 180,E1 -23977.754,E2 -23977.754} C_VEL
LIN {X 0,Y 158.494,Z 460.52,A -85,B 0,C 180,E1 -23981.081,E2 -23981.081} C_VEL
LIN {X 0,Y 154.72,Z 465.633,A -85,B 0,C 180,E1 -23985.249,E2 -23985.249} C_VEL
LIN {X 0,Y 151.707,Z 469.352,A -85,B 0,C 180,E1 -23989.57,E2 -23989.57} C_VEL
LIN {X 0,Y 150.068,Z 471.262,A -85,B 0,C 180,E1 -23992.746,E2 -23992.746} C_VEL
LIN {X 0,Y 148.964,Z 472.443,A -85,B 0,C 180,E1 -23995.521,E2 -23995.521} C_VEL
LIN {X 0,Y 148.045,Z 473.221,A -85,B 0,C 180,E1 -23998.683,E2 -23998.683} C_VEL
LIN {X 0,Y 147.444,Z 473.497,A -85,B 0,C 180,E1 -24001.536,E2 -24001.536} C_VEL
LIN {X 0,Y 147.053,Z 473.191,A -85,B 0,C 180,E1 -24005.211,E2 -24005.211} C_VEL
LIN {X 0,Y 147.163,Z 471.538,A -85,B 0,C 180,E1 -24010.473,E2 -24010.473} C_VEL
LIN {X 0,Y 147.833,Z 468.98,A -85,B 0,C 180,E1 -24014.845,E2 -24014.845} C_VEL
LIN {X 0,Y 148.967,Z 465.332,A -85,B 0,C 180,E1 -24019.125,E2 -24019.125} C_VEL
LIN {X 0,Y 150.589,Z 460.499,A -85,B 0,C 180,E1 -24023.302,E2 -24023.302} C_VEL
LIN {X 0,Y 152.799,Z 454.327,A -85,B 0,C 180,E1 -24027.366,E2 -24027.366} C_VEL
LIN {X 0,Y 155.703,Z 446.591,A -85,B 0,C 180,E1 -24031.295,E2 -24031.295} C_VEL
LIN {X 0,Y 158.54,Z 438.684,A -85,B 0,C 180,E1 -24034.451,E2 -24034.451} C_VEL
LIN {X 0,Y 161.866,Z 428.985,A -85,B 0,C 180,E1 -24037.486,E2 -24037.486} C_VEL
LIN {X 0,Y 165.226,Z 418.127,A -85,B 0,C 180,E1 -24040.107,E2 -24040.107} C_VEL
LIN {X 0,Y 168.429,Z 405.996,A -85,B 0,C 180,E1 -24042.35,E2 -24042.35} C_VEL
LIN {X 0,Y 171.048,Z 393.069,A -85,B 0,C 180,E1 -24044.122,E2 -24044.122} C_VEL
LIN {X 0,Y 173.191,Z 379.96,A -85,B 0,C 180,E1 -24045.371,E2 -24045.371} C_VEL
LIN {X 0,Y 174.622,Z 367.041,A -85,B 0,C 180,E1 -24046.14,E2 -24046.14} C_VEL
LIN {X 0,Y 177.384,Z 320.364,A -85,B 0,C 180,E1 -24047.96,E2 -24047.96} C_VEL
LIN {X 0,Y 173.345,Z 309.151,A -85,B 0,C 180,E1 -24049.514,E2 -24049.514} C_VEL
LIN {X 0,Y 167.978,Z 297.29,A -85,B 0,C 180,E1 -24051.541,E2 -24051.541} C_VEL
LIN {X 0,Y 162.355,Z 287.637,A -85,B 0,C 180,E1 -24053.705,E2 -24053.705} C_VEL
LIN {X 0,Y 157.334,Z 279.856,A -85,B 0,C 180,E1 -24055.771,E2 -24055.771} C_VEL
LIN {X 0,Y 155.43,Z 276.86,A -85,B 0,C 180,E1 -24056.599,E2 -24056.599} C_VEL
LIN {X 0,Y 153.273,Z 273.534,A -85,B 0,C 180,E1 -24057.568,E2 -24057.568} C_VEL
LIN {X 0,Y 150.885,Z 270.538,A -85,B 0,C 180,E1 -24058.646,E2 -24058.646} C_VEL
LIN {X 0,Y 150.287,Z 268.81,A -85,B 0,C 180,E1 -24059.262,E2 -24059.262} C_VEL
LIN {X 0,Y 150.172,Z 268.322,A -85,B 0,C 180,E1 -24059.821,E2 -24059.821} C_VEL
LIN {X 0,Y 150.166,Z 268.258,A -85,B 0,C 180,E1 -24064.17,E2 -24064.17} C_VEL
LIN {X 0,Y 150.157,Z 268.269,A -85,B 0,C 180,E1 -24067.48,E2 -24067.48} C_VEL
LIN {X 0,Y 150.114,Z 268.257,A -85,B 0,C 180,E1 -24071.505,E2 -24071.505} C_VEL
LIN {X 0,Y 150.11,Z 268.276,A -85,B 0,C 180,E1 -24075.404,E2 -24075.404} C_VEL
LIN {X 0,Y 150.121,Z 268.257,A -85,B 0,C 180,E1 -24079.063,E2 -24079.063} C_VEL
LIN {X 0,Y 150.162,Z 268.243,A -85,B 0,C 180,E1 -24082.719,E2 -24082.719} C_VEL
LIN {X 0,Y 150.191,Z 268.266,A -85,B 0,C 180,E1 -24087.386,E2 -24087.386} C_VEL
LIN {X 0,Y 150.173,Z 268.233,A -85,B 0,C 180,E1 -24092.775,E2 -24092.775} C_VEL
LIN {X 0,Y 150.278,Z 268.237,A -85,B 0,C 180,E1 -24099.287,E2 -24099.287} C_VEL
LIN {X 0,Y 150.319,Z 268.207,A -85,B 0,C 180,E1 -24103.719,E2 -24103.719} C_VEL
LIN {X 0,Y 150.607,Z 268.219,A -85,B 0,C 180,E1 -24109.252,E2 -24109.252} C_VEL
LIN {X 0,Y 150.681,Z 268.17,A -85,B 0,C 180,E1 -24111.966,E2 -24111.966} C_VEL
LIN {X 0,Y 151.2,Z 268.149,A -85,B 0,C 180,E1 -24120.009,E2 -24120.009} C_VEL
LIN {X 0,Y 150.691,Z 268.186,A -85,B 0,C 180,E1 -24128.052,E2 -24128.052} C_VEL
LIN {X 0,Y 150.584,Z 268.223,A -85,B 0,C 180,E1 -24131.44,E2 -24131.44} C_VEL
LIN {X 0,Y 150.34,Z 268.218,A -85,B 0,C 180,E1 -24136.298,E2 -24136.298} C_VEL
LIN {X 0,Y 150.351,Z 268.252,A -85,B 0,C 180,E1 -24140.787,E2 -24140.787} C_VEL
LIN {X 0,Y 150.253,Z 268.265,A -85,B 0,C 180,E1 -24147.284,E2 -24147.284} C_VEL
LIN {X 0,Y 150.22,Z 268.252,A -85,B 0,C 180,E1 -24152.631,E2 -24152.631} C_VEL
LIN {X 0,Y 150.223,Z 268.419,A -85,B 0,C 180,E1 -24157.242,E2 -24157.242} C_VEL
LIN {X 0,Y 150.47,Z 269.622,A -85,B 0,C 180,E1 -24157.925,E2 -24157.925} C_VEL
LIN {X 0,Y 152.184,Z 272.367,A -85,B 0,C 180,E1 -24158.79,E2 -24158.79} C_VEL
LIN {X 0,Y 153.32,Z 273.764,A -85,B 0,C 180,E1 -24159.293,E2 -24159.293} C_VEL
LIN {X 0,Y 155.489,Z 277.05,A -85,B 0,C 180,E1 -24160.261,E2 -24160.261} C_VEL
LIN {X 0,Y 160.746,Z 285.292,A -85,B 0,C 180,E1 -24162.492,E2 -24162.492} C_VEL
LIN {X 0,Y 166.769,Z 297.399,A -85,B 0,C 180,E1 -24164.966,E2 -24164.966} C_VEL
LIN {X 0,Y 172.318,Z 310.493,A -85,B 0,C 180,E1 -24167.136,E2 -24167.136} C_VEL
LIN {X 0,Y 177.262,Z 323.998,A -85,B 0,C 180,E1 -24169.03,E2 -24169.03} C_VEL
LIN {X 0,Y 174.245,Z 374.349,A -85,B 0,C 180,E1 -24171.035,E2 -24171.035} C_VEL
LIN {X 0,Y 172.475,Z 388.16,A -85,B 0,C 180,E1 -24171.988,E2 -24171.988} C_VEL
LIN {X 0,Y 170.267,Z 400.239,A -85,B 0,C 180,E1 -24173.235,E2 -24173.235} C_VEL
LIN {X 0,Y 167.733,Z 411.356,A -85,B 0,C 180,E1 -24174.819,E2 -24174.819} C_VEL
LIN {X 0,Y 164.569,Z 422.965,A -85,B 0,C 180,E1 -24177.008,E2 -24177.008} C_VEL
LIN {X 0,Y 161.259,Z 433.421,A -85,B 0,C 180,E1 -24179.558,E2 -24179.558} C_VEL
LIN {X 0,Y 158.317,Z 442.33,A -85,B 0,C 180,E1 -24182.359,E2 -24182.359} C_VEL
LIN {X 0,Y 155.18,Z 451.238,A -85,B 0,C 180,E1 -24185.943,E2 -24185.943} C_VEL
LIN {X 0,Y 152.236,Z 459.032,A -85,B 0,C 180,E1 -24189.98,E2 -24189.98} C_VEL
LIN {X 0,Y 150.185,Z 464.594,A -85,B 0,C 180,E1 -24193.691,E2 -24193.691} C_VEL
LIN {X 0,Y 148.802,Z 469.266,A -85,B 0,C 180,E1 -24197.727,E2 -24197.727} C_VEL
LIN {X 0,Y 148.16,Z 471.765,A -85,B 0,C 180,E1 -24200.493,E2 -24200.493} C_VEL
LIN {X 0,Y 147.141,Z 473.395,A -85,B 0,C 180,E1 -24202.666,E2 -24202.666} C_VEL
LIN {X 0,Y 143.989,Z 475.423,A -85,B 0,C 180,E1 -24206.282,E2 -24206.282} C_VEL
LIN {X 0,Y 141.512,Z 476.498,A -85,B 0,C 180,E1 -24209.311,E2 -24209.311} C_VEL
LIN {X 0,Y 140.504,Z 477.046,A -85,B 0,C 180,E1 -24211.695,E2 -24211.695} C_VEL
LIN {X 0,Y 140.439,Z 477.161,A -85,B 0,C 180,E1 -24212.504,E2 -24212.504} C_VEL
LIN {X 0,Y 140.573,Z 477.407,A -85,B 0,C 180,E1 -24215.736,E2 -24215.736} C_VEL
LIN {X 0,Y 141.567,Z 476.531,A -85,B 0,C 180,E1 -24221.451,E2 -24221.451} C_VEL
LIN {X 0,Y 143.698,Z 474.126,A -85,B 0,C 180,E1 -24227.062,E2 -24227.062} C_VEL
LIN {X 0,Y 146.127,Z 471.209,A -85,B 0,C 180,E1 -24231.141,E2 -24231.141} C_VEL
LIN {X 0,Y 149.401,Z 467.279,A -85,B 0,C 180,E1 -24235.045,E2 -24235.045} C_VEL
LIN {X 0,Y 153.145,Z 462.259,A -85,B 0,C 180,E1 -24238.804,E2 -24238.804} C_VEL
LIN {X 0,Y 157.532,Z 455.993,A -85,B 0,C 180,E1 -24242.365,E2 -24242.365} C_VEL
LIN {X 0,Y 162.545,Z 448.183,A -85,B 0,C 180,E1 -24245.708,E2 -24245.708} C_VEL
LIN {X 0,Y 168.213,Z 438.49,A -85,B 0,C 180,E1 -24248.805,E2 -24248.805} C_VEL
LIN {X 0,Y 173.25,Z 428.461,A -85,B 0,C 180,E1 -24251.235,E2 -24251.235} C_VEL
LIN {X 0,Y 178.109,Z 417.166,A -85,B 0,C 180,E1 -24253.28,E2 -24253.28} C_VEL
LIN {X 0,Y 182.035,Z 406.139,A -85,B 0,C 180,E1 -24254.794,E2 -24254.794} C_VEL
LIN {X 0,Y 185.429,Z 393.919,A -85,B 0,C 180,E1 -24256.062,E2 -24256.062} C_VEL
LIN {X 0,Y 188.201,Z 380.628,A -85,B 0,C 180,E1 -24256.974,E2 -24256.974} C_VEL
LIN {X 0,Y 189.862,Z 367.593,A -85,B 0,C 180,E1 -24257.569,E2 -24257.569} C_VEL
LIN {X 0,Y 192.169,Z 339.189,A -85,B 0,C 180,E1 -24258.543,E2 -24258.543} C_VEL
LIN {X 0,Y 188.487,Z 329.648,A -85,B 0,C 180,E1 -24260.959,E2 -24260.959} C_VEL
LIN {X 0,Y 184.416,Z 320.895,A -85,B 0,C 180,E1 -24263.847,E2 -24263.847} C_VEL
LIN {X 0,Y 181.242,Z 314.789,A -85,B 0,C 180,E1 -24266.382,E2 -24266.382} C_VEL
LIN {X 0,Y 177.651,Z 308.338,A -85,B 0,C 180,E1 -24269.724,E2 -24269.724} C_VEL
LIN {X 0,Y 174.946,Z 304.423,A -85,B 0,C 180,E1 -24272.639,E2 -24272.639} C_VEL
LIN {X 0,Y 172.11,Z 300.904,A -85,B 0,C 180,E1 -24276.494,E2 -24276.494} C_VEL
LIN {X 0,Y 171.318,Z 299.191,A -85,B 0,C 180,E1 -24277.957,E2 -24277.957} C_VEL
LIN {X 0,Y 168.449,Z 295.692,A -85,B 0,C 180,E1 -24287.951,E2 -24287.951} C_VEL
LIN {X 0,Y 168.582,Z 295.688,A -85,B 0,C 180,E1 -24290.778,E2 -24290.778} C_VEL
LIN {X 0,Y 171.606,Z 299.039,A -85,B 0,C 180,E1 -24299.699,E2 -24299.699} C_VEL
LIN {X 0,Y 173.351,Z 302.353,A -85,B 0,C 180,E1 -24302.554,E2 -24302.554} C_VEL
LIN {X 0,Y 175.164,Z 304.292,A -85,B 0,C 180,E1 -24304.808,E2 -24304.808} C_VEL
LIN {X 0,Y 178.43,Z 309.271,A -85,B 0,C 180,E1 -24308.254,E2 -24308.254} C_VEL
LIN {X 0,Y 181.408,Z 313.979,A -85,B 0,C 180,E1 -24310.896,E2 -24310.896} C_VEL
LIN {X 0,Y 185.015,Z 319.729,A -85,B 0,C 180,E1 -24313.643,E2 -24313.643} C_VEL
LIN {X 0,Y 188.926,Z 327.85,A -85,B 0,C 180,E1 -24316.365,E2 -24316.365} C_VEL
LIN {X 0,Y 192.395,Z 336.337,A -85,B 0,C 180,E1 -24318.602,E2 -24318.602} C_VEL
LIN {X 0,Y 189.393,Z 370.79,A -85,B 0,C 180,E1 -24319.8,E2 -24319.8} C_VEL
LIN {X 0,Y 187.333,Z 383.308,A -85,B 0,C 180,E1 -24320.497,E2 -24320.497} C_VEL
LIN {X 0,Y 184.246,Z 396.457,A -85,B 0,C 180,E1 -24321.606,E2 -24321.606} C_VEL
LIN {X 0,Y 180.742,Z 408.091,A -85,B 0,C 180,E1 -24323.04,E2 -24323.04} C_VEL
LIN {X 0,Y 176.256,Z 419.707,A -85,B 0,C 180,E1 -24324.894,E2 -24324.894} C_VEL
LIN {X 0,Y 171.451,Z 430.191,A -85,B 0,C 180,E1 -24327.109,E2 -24327.109} C_VEL
LIN {X 0,Y 166.117,Z 440.044,A -85,B 0,C 180,E1 -24329.861,E2 -24329.861} C_VEL
LIN {X 0,Y 161.102,Z 448.275,A -85,B 0,C 180,E1 -24332.888,E2 -24332.888} C_VEL
LIN {X 0,Y 156.559,Z 454.987,A -85,B 0,C 180,E1 -24336.101,E2 -24336.101} C_VEL
LIN {X 0,Y 152.33,Z 460.79,A -85,B 0,C 180,E1 -24339.753,E2 -24339.753} C_VEL
LIN {X 0,Y 149.084,Z 464.816,A -85,B 0,C 180,E1 -24343.059,E2 -24343.059} C_VEL
LIN {X 0,Y 145.718,Z 468.828,A -85,B 0,C 180,E1 -24347.532,E2 -24347.532} C_VEL
LIN {X 0,Y 143.402,Z 471.307,A -85,B 0,C 180,E1 -24351.624,E2 -24351.624} C_VEL
LIN {X 0,Y 141.393,Z 473.144,A -85,B 0,C 180,E1 -24356.858,E2 -24356.858} C_VEL
LIN {X 0,Y 140.619,Z 473.552,A -85,B 0,C 180,E1 -24360.017,E2 -24360.017} C_VEL
LIN {X 0,Y 140.013,Z 473.328,A -85,B 0,C 180,E1 -24364.597,E2 -24364.597} C_VEL
LIN {X 0,Y 139.972,Z 472.001,A -85,B 0,C 180,E1 -24369.426,E2 -24369.426} C_VEL
LIN {X 0,Y 140.322,Z 470.561,A -85,B 0,C 180,E1 -24372.514,E2 -24372.514} C_VEL
LIN {X 0,Y 141.222,Z 467.501,A -85,B 0,C 180,E1 -24377.062,E2 -24377.062} C_VEL
LIN {X 0,Y 142.663,Z 463.317,A -85,B 0,C 180,E1 -24381.504,E2 -24381.504} C_VEL
LIN {X 0,Y 145.018,Z 456.83,A -85,B 0,C 180,E1 -24386.529,E2 -24386.529} C_VEL
LIN {X 0,Y 147.807,Z 449.698,A -85,B 0,C 180,E1 -24390.696,E2 -24390.696} C_VEL
LIN {X 0,Y 150.626,Z 442.433,A -85,B 0,C 180,E1 -24394.015,E2 -24394.015} C_VEL
LIN {X 0,Y 154.228,Z 432.567,A -85,B 0,C 180,E1 -24397.53,E2 -24397.53} C_VEL
LIN {X 0,Y 157.588,Z 422.58,A -85,B 0,C 180,E1 -24400.278,E2 -24400.278} C_VEL
LIN {X 0,Y 160.857,Z 411.605,A -85,B 0,C 180,E1 -24402.62,E2 -24402.62} C_VEL
LIN {X 0,Y 163.813,Z 399.319,A -85,B 0,C 180,E1 -24404.601,E2 -24404.601} C_VEL
LIN {X 0,Y 166.267,Z 386.49,A -85,B 0,C 180,E1 -24406.107,E2 -24406.107} C_VEL
LIN {X 0,Y 168.028,Z 373.999,A -85,B 0,C 180,E1 -24407.098,E2 -24407.098} C_VEL
LIN {X 0,Y 169.329,Z 358.482,A -85,B 0,C 180,E1 -24407.819,E2 -24407.819} C_VEL
LIN {X 0,Y 171.578,Z 322.464,A -85,B 0,C 180,E1 -24409.226,E2 -24409.226} C_VEL
LIN {X 0,Y 168.373,Z 313.206,A -85,B 0,C 180,E1 -24410.538,E2 -24410.538} C_VEL
LIN {X 0,Y 163.021,Z 301.18,A -85,B 0,C 180,E1 -24412.698,E2 -24412.698} C_VEL
LIN {X 0,Y 157.706,Z 291.956,A -85,B 0,C 180,E1 -24414.879,E2 -24414.879} C_VEL
LIN {X 0,Y 151.41,Z 282.029,A -85,B 0,C 180,E1 -24417.659,E2 -24417.659} C_VEL
LIN {X 0,Y 148.488,Z 277.837,A -85,B 0,C 180,E1 -24419.042,E2 -24419.042} C_VEL
LIN {X 0,Y 146.403,Z 274.625,A -85,B 0,C 180,E1 -24420.1,E2 -24420.1} C_VEL
LIN {X 0,Y 143.805,Z 271.399,A -85,B 0,C 180,E1 -24421.433,E2 -24421.433} C_VEL
LIN {X 0,Y 143.217,Z 269.698,A -85,B 0,C 180,E1 -24422.067,E2 -24422.067} C_VEL
LIN {X 0,Y 143.154,Z 269.194,A -85,B 0,C 180,E1 -24422.688,E2 -24422.688} C_VEL
LIN {X 0,Y 143.059,Z 269.162,A -85,B 0,C 180,E1 -24428.202,E2 -24428.202} C_VEL
LIN {X 0,Y 143.015,Z 269.139,A -85,B 0,C 180,E1 -24433.473,E2 -24433.473} C_VEL
LIN {X 0,Y 143.04,Z 269.162,A -85,B 0,C 180,E1 -24437.479,E2 -24437.479} C_VEL
LIN {X 0,Y 143.057,Z 269.122,A -85,B 0,C 180,E1 -24441.82,E2 -24441.82} C_VEL
LIN {X 0,Y 143.159,Z 269.142,A -85,B 0,C 180,E1 -24447.328,E2 -24447.328} C_VEL
LIN {X 0,Y 143.097,Z 269.124,A -85,B 0,C 180,E1 -24453.779,E2 -24453.779} C_VEL
LIN {X 0,Y 143.243,Z 269.101,A -85,B 0,C 180,E1 -24459.924,E2 -24459.924} C_VEL
LIN {X 0,Y 143.312,Z 269.104,A -85,B 0,C 180,E1 -24465.817,E2 -24465.817} C_VEL
LIN {X 0,Y 143.533,Z 269.104,A -85,B 0,C 180,E1 -24468.715,E2 -24468.715} C_VEL
LIN {X 0,Y 143.607,Z 269.055,A -85,B 0,C 180,E1 -24471.567,E2 -24471.567} C_VEL
LIN {X 0,Y 144.159,Z 269.026,A -85,B 0,C 180,E1 -24480.009,E2 -24480.009} C_VEL
LIN {X 0,Y 143.617,Z 269.072,A -85,B 0,C 180,E1 -24488.451,E2 -24488.451} C_VEL
LIN {X 0,Y 143.51,Z 269.101,A -85,B 0,C 180,E1 -24491.629,E2 -24491.629} C_VEL
LIN {X 0,Y 143.279,Z 269.103,A -85,B 0,C 180,E1 -24497.125,E2 -24497.125} C_VEL
LIN {X 0,Y 143.279,Z 269.124,A -85,B 0,C 180,E1 -24501.251,E2 -24501.251} C_VEL
LIN {X 0,Y 143.197,Z 269.149,A -85,B 0,C 180,E1 -24507.937,E2 -24507.937} C_VEL
LIN {X 0,Y 143.186,Z 269.213,A -85,B 0,C 180,E1 -24514.254,E2 -24514.254} C_VEL
LIN {X 0,Y 143.437,Z 270.358,A -85,B 0,C 180,E1 -24515.099,E2 -24515.099} C_VEL
LIN {X 0,Y 145.139,Z 273.146,A -85,B 0,C 180,E1 -24516.099,E2 -24516.099} C_VEL
LIN {X 0,Y 146.413,Z 274.686,A -85,B 0,C 180,E1 -24516.739,E2 -24516.739} C_VEL
LIN {X 0,Y 148.632,Z 278.013,A -85,B 0,C 180,E1 -24517.856,E2 -24517.856} C_VEL
LIN {X 0,Y 154.852,Z 287.504,A -85,B 0,C 180,E1 -24520.734,E2 -24520.734} C_VEL
LIN {X 0,Y 158.827,Z 294.947,A -85,B 0,C 180,E1 -24522.493,E2 -24522.493} C_VEL
LIN {X 0,Y 164.464,Z 307.25,A -85,B 0,C 180,E1 -24524.901,E2 -24524.901} C_VEL
LIN {X 0,Y 170.928,Z 324.307,A -85,B 0,C 180,E1 -24527.545,E2 -24527.545} C_VEL
LIN {X 0,Y 171.476,Z 325.946,A -85,B 0,C 180,E1 -24527.766,E2 -24527.766} C_VEL
LIN {X 0,Y 168.304,Z 374.69,A -85,B 0,C 180,E1 -24529.739,E2 -24529.739} C_VEL
LIN {X 0,Y 166.481,Z 388.312,A -85,B 0,C 180,E1 -24530.709,E2 -24530.709} C_VEL
LIN {X 0,Y 164.145,Z 400.521,A -85,B 0,C 180,E1 -24532.011,E2 -24532.011} C_VEL
LIN {X 0,Y 161.098,Z 413.139,A -85,B 0,C 180,E1 -24533.916,E2 -24533.916} C_VEL
LIN {X 0,Y 157.795,Z 424.398,A -85,B 0,C 180,E1 -24536.167,E2 -24536.167} C_VEL
LIN {X 0,Y 154.451,Z 434.538,A -85,B 0,C 180,E1 -24538.827,E2 -24538.827} C_VEL
LIN {X 0,Y 150.804,Z 444.756,A -85,B 0,C 180,E1 -24542.325,E2 -24542.325} C_VEL
LIN {X 0,Y 148.126,Z 451.952,A -85,B 0,C 180,E1 -24545.469,E2 -24545.469} C_VEL
LIN {X 0,Y 145.262,Z 459.228,A -85,B 0,C 180,E1 -24549.464,E2 -24549.464} C_VEL
LIN {X 0,Y 143.348,Z 464.123,A -85,B 0,C 180,E1 -24552.89,E2 -24552.89} C_VEL
LIN {X 0,Y 141.832,Z 468.874,A -85,B 0,C 180,E1 -24557.113,E2 -24557.113} C_VEL
LIN {X 0,Y 140.888,Z 472.48,A -85,B 0,C 180,E1 -24561.391,E2 -24561.391} C_VEL
LIN {X 0,Y 140.569,Z 474.322,A -85,B 0,C 180,E1 -24564.259,E2 -24564.259} C_VEL
LIN {X 0,Y 140.449,Z 475.693,A -85,B 0,C 180,E1 -24567.129,E2 -24567.129} C_VEL
LIN {X 0,Y 140.521,Z 476.662,A -85,B 0,C 180,E1 -24569.998,E2 -24569.998} C_VEL
LIN {X 0,Y 140.439,Z 477.161,A -85,B 0,C 180,E1 -24572.504,E2 -24572.504} C_VEL
LIN {X 0,Y 139.882,Z 477.477,A -85,B 0,C 180,E1 -24574.902,E2 -24574.902} C_VEL
LIN {X 0,Y 137.497,Z 477.318,A -85,B 0,C 180,E1 -24578.879,E2 -24578.879} C_VEL
LIN {X 0,Y 135.795,Z 476.594,A -85,B 0,C 180,E1 -24582.142,E2 -24582.142} C_VEL
LIN {X 0,Y 135.54,Z 475.711,A -85,B 0,C 180,E1 -24584.626,E2 -24584.626} C_VEL
LIN {X 0,Y 135.768,Z 475.352,A -85,B 0,C 180,E1 -24585.445,E2 -24585.445} C_VEL
LIN {X 0,Y 138.513,Z 472.421,A -85,B 0,C 180,E1 -24590.801,E2 -24590.801} C_VEL
LIN {X 0,Y 141.756,Z 468.935,A -85,B 0,C 180,E1 -24594.921,E2 -24594.921} C_VEL
LIN {X 0,Y 145.552,Z 464.391,A -85,B 0,C 180,E1 -24598.869,E2 -24598.869} C_VEL
LIN {X 0,Y 150.695,Z 457.659,A -85,B 0,C 180,E1 -24603.146,E2 -24603.146} C_VEL
LIN {X 0,Y 155.981,Z 450.168,A -85,B 0,C 180,E1 -24606.653,E2 -24606.653} C_VEL
LIN {X 0,Y 160.793,Z 442.665,A -85,B 0,C 180,E1 -24609.326,E2 -24609.326} C_VEL
LIN {X 0,Y 164.822,Z 435.553,A -85,B 0,C 180,E1 -24611.367,E2 -24611.367} C_VEL
LIN {X 0,Y 169.727,Z 426.013,A -85,B 0,C 180,E1 -24613.501,E2 -24613.501} C_VEL
LIN {X 0,Y 174.214,Z 415.665,A -85,B 0,C 180,E1 -24615.314,E2 -24615.314} C_VEL
LIN {X 0,Y 178.313,Z 404.283,A -85,B 0,C 180,E1 -24616.812,E2 -24616.812} C_VEL
LIN {X 0,Y 181.83,Z 391.541,A -85,B 0,C 180,E1 -24618.048,E2 -24618.048} C_VEL
LIN {X 0,Y 184.609,Z 378.001,A -85,B 0,C 180,E1 -24618.906,E2 -24618.906} C_VEL
LIN {X 0,Y 186.276,Z 363.054,A -85,B 0,C 180,E1 -24619.514,E2 -24619.514} C_VEL
LIN {X 0,Y 188.047,Z 341.916,A -85,B 0,C 180,E1 -24620.245,E2 -24620.245} C_VEL
LIN {X 0,Y 184.861,Z 333.446,A -85,B 0,C 180,E1 -24622.527,E2 -24622.527} C_VEL
LIN {X 0,Y 181.196,Z 325.318,A -85,B 0,C 180,E1 -24625.408,E2 -24625.408} C_VEL
LIN {X 0,Y 178.382,Z 319.564,A -85,B 0,C 180,E1 -24627.897,E2 -24627.897} C_VEL
LIN {X 0,Y 175.661,Z 314.598,A -85,B 0,C 180,E1 -24630.659,E2 -24630.659} C_VEL
LIN {X 0,Y 173.121,Z 310.728,A -85,B 0,C 180,E1 -24633.643,E2 -24633.643} C_VEL
LIN {X 0,Y 170.774,Z 307.697,A -85,B 0,C 180,E1 -24637.059,E2 -24637.059} C_VEL
LIN {X 0,Y 170.016,Z 306.049,A -85,B 0,C 180,E1 -24638.58,E2 -24638.58} C_VEL
LIN {X 0,Y 167.515,Z 302.765,A -85,B 0,C 180,E1 -24647.883,E2 -24647.883} C_VEL
LIN {X 0,Y 167.639,Z 302.748,A -85,B 0,C 180,E1 -24650.725,E2 -24650.725} C_VEL
LIN {X 0,Y 170.3,Z 305.899,A -85,B 0,C 180,E1 -24659.105,E2 -24659.105} C_VEL
LIN {X 0,Y 172.053,Z 309.201,A -85,B 0,C 180,E1 -24662.128,E2 -24662.128} C_VEL
LIN {X 0,Y 173.62,Z 311.025,A -85,B 0,C 180,E1 -24664.181,E2 -24664.181} C_VEL
LIN {X 0,Y 176.534,Z 315.699,A -85,B 0,C 180,E1 -24667.461,E2 -24667.461} C_VEL
LIN {X 0,Y 179.171,Z 320.07,A -85,B 0,C 180,E1 -24669.981,E2 -24669.981} C_VEL
LIN {X 0,Y 182.527,Z 325.695,A -85,B 0,C 180,E1 -24672.698,E2 -24672.698} C_VEL
LIN {X 0,Y 185.847,Z 333.074,A -85,B 0,C 180,E1 -24675.214,E2 -24675.214} C_VEL
LIN {X 0,Y 188.287,Z 339.371,A -85,B 0,C 180,E1 -24676.925,E2 -24676.925} C_VEL
LIN {X 0,Y 185.348,Z 371.217,A -85,B 0,C 180,E1 -24678.028,E2 -24678.028} C_VEL
LIN {X 0,Y 183.185,Z 383.694,A -85,B 0,C 180,E1 -24678.718,E2 -24678.718} C_VEL
LIN {X 0,Y 180.16,Z 396.134,A -85,B 0,C 180,E1 -24679.768,E2 -24679.768} C_VEL
LIN {X 0,Y 176.597,Z 407.516,A -85,B 0,C 180,E1 -24681.131,E2 -24681.131} C_VEL
LIN {X 0,Y 171.825,Z 419.49,A -85,B 0,C 180,E1 -24683.037,E2 -24683.037} C_VEL
LIN {X 0,Y 167.375,Z 428.803,A -85,B 0,C 180,E1 -24684.963,E2 -24684.963} C_VEL
LIN {X 0,Y 162.316,Z 438.056,A -85,B 0,C 180,E1 -24687.43,E2 -24687.43} C_VEL
LIN {X 0,Y 156.901,Z 446.688,A -85,B 0,C 180,E1 -24690.448,E2 -24690.448} C_VEL
LIN {X 0,Y 151.952,Z 453.739,A -85,B 0,C 180,E1 -24693.7,E2 -24693.7} C_VEL
LIN {X 0,Y 146.911,Z 460.273,A -85,B 0,C 180,E1 -24697.727,E2 -24697.727} C_VEL
LIN {X 0,Y 142.367,Z 465.593,A -85,B 0,C 180,E1 -24702.232,E2 -24702.232} C_VEL
LIN {X 0,Y 138.832,Z 469.388,A -85,B 0,C 180,E1 -24706.894,E2 -24706.894} C_VEL
LIN {X 0,Y 136.149,Z 471.941,A -85,B 0,C 180,E1 -24711.728,E2 -24711.728} C_VEL
LIN {X 0,Y 134.238,Z 473.384,A -85,B 0,C 180,E1 -24716.874,E2 -24716.874} C_VEL
LIN {X 0,Y 133.209,Z 473.669,A -85,B 0,C 180,E1 -24721.655,E2 -24721.655} C_VEL
LIN {X 0,Y 132.883,Z 473.29,A -85,B 0,C 180,E1 -24724.972,E2 -24724.972} C_VEL
LIN {X 0,Y 132.821,Z 472.458,A -85,B 0,C 180,E1 -24728.263,E2 -24728.263} C_VEL
LIN {X 0,Y 133.117,Z 470.975,A -85,B 0,C 180,E1 -24731.825,E2 -24731.825} C_VEL
LIN {X 0,Y 133.914,Z 468.259,A -85,B 0,C 180,E1 -24736.342,E2 -24736.342} C_VEL
LIN {X 0,Y 135.332,Z 464.286,A -85,B 0,C 180,E1 -24741.04,E2 -24741.04} C_VEL
LIN {X 0,Y 137.257,Z 459.119,A -85,B 0,C 180,E1 -24745.598,E2 -24745.598} C_VEL
LIN {X 0,Y 139.944,Z 452.572,A -85,B 0,C 180,E1 -24750.002,E2 -24750.002} C_VEL
LIN {X 0,Y 143.277,Z 444.318,A -85,B 0,C 180,E1 -24754.222,E2 -24754.222} C_VEL
LIN {X 0,Y 146.553,Z 435.867,A -85,B 0,C 180,E1 -24757.58,E2 -24757.58} C_VEL
LIN {X 0,Y 150.388,Z 425.465,A -85,B 0,C 180,E1 -24760.776,E2 -24760.776} C_VEL
LIN {X 0,Y 153.728,Z 415.088,A -85,B 0,C 180,E1 -24763.216,E2 -24763.216} C_VEL
LIN {X 0,Y 156.765,Z 403.808,A -85,B 0,C 180,E1 -24765.273,E2 -24765.273} C_VEL
LIN {X 0,Y 159.46,Z 391.341,A -85,B 0,C 180,E1 -24766.979,E2 -24766.979} C_VEL
LIN {X 0,Y 161.641,Z 378.214,A -85,B 0,C 180,E1 -24768.197,E2 -24768.197} C_VEL
LIN {X 0,Y 163.089,Z 364.787,A -85,B 0,C 180,E1 -24768.975,E2 -24768.975} C_VEL
LIN {X 0,Y 165.707,Z 323.696,A -85,B 0,C 180,E1 -24770.642,E2 -24770.642} C_VEL
LIN {X 0,Y 161.8,Z 313.226,A -85,B 0,C 180,E1 -24772.331,E2 -24772.331} C_VEL
LIN {X 0,Y 158.024,Z 304.872,A -85,B 0,C 180,E1 -24773.969,E2 -24773.969} C_VEL
LIN {X 0,Y 153.117,Z 296.329,A -85,B 0,C 180,E1 -24776.098,E2 -24776.098} C_VEL
LIN {X 0,Y 147.24,Z 286.919,A -85,B 0,C 180,E1 -24778.874,E2 -24778.874} C_VEL
LIN {X 0,Y 143.936,Z 282.109,A -85,B 0,C 180,E1 -24780.56,E2 -24780.56} C_VEL
LIN {X 0,Y 142.034,Z 279.295,A -85,B 0,C 180,E1 -24781.582,E2 -24781.582} C_VEL
LIN {X 0,Y 139.706,Z 275.961,A -85,B 0,C 180,E1 -24782.879,E2 -24782.879} C_VEL
LIN {X 0,Y 139.089,Z 274.987,A -85,B 0,C 180,E1 -24783.243,E2 -24783.243} C_VEL
LIN {X 0,Y 137.023,Z 272.842,A -85,B 0,C 180,E1 -24784.409,E2 -24784.409} C_VEL
LIN {X 0,Y 136.149,Z 270.737,A -85,B 0,C 180,E1 -24785.276,E2 -24785.276} C_VEL
LIN {X 0,Y 136.044,Z 270.108,A -85,B 0,C 180,E1 -24785.99,E2 -24785.99} C_VEL
LIN {X 0,Y 136.009,Z 270.039,A -85,B 0,C 180,E1 -24789.205,E2 -24789.205} C_VEL
LIN {X 0,Y 135.961,Z 270.018,A -85,B 0,C 180,E1 -24793.658,E2 -24793.658} C_VEL
LIN {X 0,Y 135.981,Z 270.034,A -85,B 0,C 180,E1 -24797.802,E2 -24797.802} C_VEL
LIN {X 0,Y 136.006,Z 270,A -85,B 0,C 180,E1 -24801.692,E2 -24801.692} C_VEL
LIN {X 0,Y 136.039,Z 270.038,A -85,B 0,C 180,E1 -24805.753,E2 -24805.753} C_VEL
LIN {X 0,Y 136.074,Z 269.984,A -85,B 0,C 180,E1 -24812.313,E2 -24812.313} C_VEL
LIN {X 0,Y 136.177,Z 269.997,A -85,B 0,C 180,E1 -24818.834,E2 -24818.834} C_VEL
LIN {X 0,Y 136.228,Z 269.973,A -85,B 0,C 180,E1 -24825.063,E2 -24825.063} C_VEL
LIN {X 0,Y 136.425,Z 269.991,A -85,B 0,C 180,E1 -24828.188,E2 -24828.188} C_VEL
LIN {X 0,Y 136.537,Z 269.94,A -85,B 0,C 180,E1 -24831.127,E2 -24831.127} C_VEL
LIN {X 0,Y 137.116,Z 269.903,A -85,B 0,C 180,E1 -24840.01,E2 -24840.01} C_VEL
LIN {X 0,Y 136.546,Z 269.959,A -85,B 0,C 180,E1 -24848.892,E2 -24848.892} C_VEL
LIN {X 0,Y 136.425,Z 269.977,A -85,B 0,C 180,E1 -24851.902,E2 -24851.902} C_VEL
LIN {X 0,Y 136.199,Z 269.995,A -85,B 0,C 180,E1 -24858.045,E2 -24858.045} C_VEL
LIN {X 0,Y 136.202,Z 269.997,A -85,B 0,C 180,E1 -24861.746,E2 -24861.746} C_VEL
LIN {X 0,Y 136.106,Z 270.023,A -85,B 0,C 180,E1 -24868.616,E2 -24868.616} C_VEL
LIN {X 0,Y 136.089,Z 270.216,A -85,B 0,C 180,E1 -24871.103,E2 -24871.103} C_VEL
LIN {X 0,Y 136.45,Z 271.499,A -85,B 0,C 180,E1 -24871.985,E2 -24871.985} C_VEL
LIN {X 0,Y 138.281,Z 274.275,A -85,B 0,C 180,E1 -24873.147,E2 -24873.147} C_VEL
LIN {X 0,Y 139.652,Z 275.717,A -85,B 0,C 180,E1 -24873.904,E2 -24873.904} C_VEL
LIN {X 0,Y 142.028,Z 279.189,A -85,B 0,C 180,E1 -24875.235,E2 -24875.235} C_VEL
LIN {X 0,Y 148.34,Z 288.676,A -85,B 0,C 180,E1 -24878.501,E2 -24878.501} C_VEL
LIN {X 0,Y 152.733,Z 296.159,A -85,B 0,C 180,E1 -24880.589,E2 -24880.589} C_VEL
LIN {X 0,Y 158.266,Z 308.056,A -85,B 0,C 180,E1 -24883.135,E2 -24883.135} C_VEL
LIN {X 0,Y 163.298,Z 321.065,A -85,B 0,C 180,E1 -24885.385,E2 -24885.385} C_VEL
LIN {X 0,Y 165.633,Z 327.577,A -85,B 0,C 180,E1 -24886.388,E2 -24886.388} C_VEL
LIN {X 0,Y 162.489,Z 374.327,A -85,B 0,C 180,E1 -24888.329,E2 -24888.329} C_VEL
LIN {X 0,Y 160.606,Z 387.745,A -85,B 0,C 180,E1 -24889.284,E2 -24889.284} C_VEL
LIN {X 0,Y 158.35,Z 399.573,A -85,B 0,C 180,E1 -24890.561,E2 -24890.561} C_VEL
LIN {X 0,Y 155.371,Z 411.612,A -85,B 0,C 180,E1 -24892.361,E2 -24892.361} C_VEL
LIN {X 0,Y 151.953,Z 423.141,A -85,B 0,C 180,E1 -24894.678,E2 -24894.678} C_VEL
LIN {X 0,Y 148.354,Z 433.53,A -85,B 0,C 180,E1 -24897.391,E2 -24897.391} C_VEL
LIN {X 0,Y 145.248,Z 442.037,A -85,B 0,C 180,E1 -24900.265,E2 -24900.265} C_VEL
LIN {X 0,Y 142.245,Z 449.871,A -85,B 0,C 180,E1 -24903.595,E2 -24903.595} C_VEL
LIN {X 0,Y 139.084,Z 457.5,A -85,B 0,C 180,E1 -24907.727,E2 -24907.727} C_VEL
LIN {X 0,Y 136.541,Z 463.615,A -85,B 0,C 180,E1 -24912.009,E2 -24912.009} C_VEL
LIN {X 0,Y 134.892,Z 468.455,A -85,B 0,C 180,E1 -24916.438,E2 -24916.438} C_VEL
LIN {X 0,Y 133.862,Z 472.143,A -85,B 0,C 180,E1 -24920.935,E2 -24920.935} C_VEL
LIN {X 0,Y 133.487,Z 474.039,A -85,B 0,C 180,E1 -24923.953,E2 -24923.953} C_VEL
LIN {X 0,Y 133.352,Z 475.468,A -85,B 0,C 180,E1 -24926.976,E2 -24926.976} C_VEL
LIN {X 0,Y 133.437,Z 476.474,A -85,B 0,C 180,E1 -24929.998,E2 -24929.998} C_VEL
LIN {X 0,Y 133.352,Z 477.08,A -85,B 0,C 180,E1 -24933.019,E2 -24933.019} C_VEL
LIN {X 0,Y 133.494,Z 477.303,A -85,B 0,C 180,E1 -24936.041,E2 -24936.041} C_VEL
LIN {X 0,Y 133.914,Z 477.113,A -85,B 0,C 180,E1 -24939.056,E2 -24939.056} C_VEL
LIN {X 0,Y 135.602,Z 475.549,A -85,B 0,C 180,E1 -24945.016,E2 -24945.016} C_VEL
LIN {X 0,Y 135.768,Z 475.352,A -85,B 0,C 180,E1 -24945.445,E2 -24945.445} C_VEL
LIN {X 0,Y 136.198,Z 474.277,A -85,B 0,C 180,E1 -24947.881,E2 -24947.881} C_VEL
LIN {X 0,Y 135.708,Z 472.031,A -85,B 0,C 180,E1 -24951.953,E2 -24951.953} C_VEL
LIN {X 0,Y 135.669,Z 469.836,A -85,B 0,C 180,E1 -24955.174,E2 -24955.174} C_VEL
LIN {X 0,Y 136.654,Z 467.845,A -85,B 0,C 180,E1 -24957.476,E2 -24957.476} C_VEL
LIN {X 0,Y 137.273,Z 467.092,A -85,B 0,C 180,E1 -24958.194,E2 -24958.194} C_VEL
LIN {X 0,Y 140.883,Z 462.938,A -85,B 0,C 180,E1 -24961.584,E2 -24961.584} C_VEL
LIN {X 0,Y 145.756,Z 456.885,A -85,B 0,C 180,E1 -24965.35,E2 -24965.35} C_VEL
LIN {X 0,Y 151.311,Z 449.407,A -85,B 0,C 180,E1 -24968.829,E2 -24968.829} C_VEL
LIN {X 0,Y 156.458,Z 441.785,A -85,B 0,C 180,E1 -24971.492,E2 -24971.492} C_VEL
LIN {X 0,Y 161.773,Z 432.572,A -85,B 0,C 180,E1 -24974.032,E2 -24974.032} C_VEL
LIN {X 0,Y 166.977,Z 422.361,A -85,B 0,C 180,E1 -24976.116,E2 -24976.116} C_VEL
LIN {X 0,Y 171.782,Z 411.094,A -85,B 0,C 180,E1 -24977.859,E2 -24977.859} C_VEL
LIN {X 0,Y 175.749,Z 399.441,A -85,B 0,C 180,E1 -24979.222,E2 -24979.222} C_VEL
LIN {X 0,Y 178.995,Z 386.874,A -85,B 0,C 180,E1 -24980.265,E2 -24980.265} C_VEL
LIN {X 0,Y 181.462,Z 373.433,A -85,B 0,C 180,E1 -24980.974,E2 -24980.974} C_VEL
LIN {X 0,Y 184.122,Z 344.723,A -85,B 0,C 180,E1 -24982.005,E2 -24982.005} C_VEL
LIN {X 0,Y 181.509,Z 337.624,A -85,B 0,C 180,E1 -24984.09,E2 -24984.09} C_VEL
LIN {X 0,Y 178.328,Z 330.214,A -85,B 0,C 180,E1 -24986.83,E2 -24986.83} C_VEL
LIN {X 0,Y 175.294,Z 323.787,A -85,B 0,C 180,E1 -24989.86,E2 -24989.86} C_VEL
LIN {X 0,Y 173.752,Z 320.928,A -85,B 0,C 180,E1 -24991.575,E2 -24991.575} C_VEL
LIN {X 0,Y 171.403,Z 317.209,A -85,B 0,C 180,E1 -24994.578,E2 -24994.578} C_VEL
LIN {X 0,Y 169.211,Z 313.901,A -85,B 0,C 180,E1 -24998.15,E2 -24998.15} C_VEL
LIN {X 0,Y 168.725,Z 312.908,A -85,B 0,C 180,E1 -24999.228,E2 -24999.228} C_VEL
LIN {X 0,Y 166.58,Z 309.843,A -85,B 0,C 180,E1 -25007.814,E2 -25007.814} C_VEL
LIN {X 0,Y 166.694,Z 309.824,A -85,B 0,C 180,E1 -25010.672,E2 -25010.672} C_VEL
LIN {X 0,Y 169.024,Z 312.716,A -85,B 0,C 180,E1 -25018.503,E2 -25018.503} C_VEL
LIN {X 0,Y 170.924,Z 316.288,A -85,B 0,C 180,E1 -25021.936,E2 -25021.936} C_VEL
LIN {X 0,Y 172.09,Z 317.751,A -85,B 0,C 180,E1 -25023.534,E2 -25023.534} C_VEL
LIN {X 0,Y 174.752,Z 322.258,A -85,B 0,C 180,E1 -25026.738,E2 -25026.738} C_VEL
LIN {X 0,Y 177.696,Z 327.333,A -85,B 0,C 180,E1 -25029.669,E2 -25029.669} C_VEL
LIN {X 0,Y 180.681,Z 332.851,A -85,B 0,C 180,E1 -25032.214,E2 -25032.214} C_VEL
LIN {X 0,Y 183.857,Z 340.772,A -85,B 0,C 180,E1 -25034.778,E2 -25034.778} C_VEL
LIN {X 0,Y 184.325,Z 342.475,A -85,B 0,C 180,E1 -25035.17,E2 -25035.17} C_VEL
LIN {X 0,Y 181.48,Z 371.723,A -85,B 0,C 180,E1 -25036.183,E2 -25036.183} C_VEL
LIN {X 0,Y 179.293,Z 383.782,A -85,B 0,C 180,E1 -25036.839,E2 -25036.839} C_VEL
LIN {X 0,Y 176.402,Z 395.319,A -85,B 0,C 180,E1 -25037.788,E2 -25037.788} C_VEL
LIN {X 0,Y 172.668,Z 407.041,A -85,B 0,C 180,E1 -25039.156,E2 -25039.156} C_VEL
LIN {X 0,Y 168.234,Z 417.931,A -85,B 0,C 180,E1 -25040.824,E2 -25040.824} C_VEL
LIN {X 0,Y 162.702,Z 429.135,A -85,B 0,C 180,E1 -25043.097,E2 -25043.097} C_VEL
LIN {X 0,Y 157.637,Z 437.974,A -85,B 0,C 180,E1 -25045.476,E2 -25045.476} C_VEL
LIN {X 0,Y 151.929,Z 446.604,A -85,B 0,C 180,E1 -25048.494,E2 -25048.494} C_VEL
LIN {X 0,Y 146.644,Z 453.704,A -85,B 0,C 180,E1 -25051.803,E2 -25051.803} C_VEL
LIN {X 0,Y 141.144,Z 460.373,A -85,B 0,C 180,E1 -25055.993,E2 -25055.993} C_VEL
LIN {X 0,Y 137.129,Z 464.802,A -85,B 0,C 180,E1 -25059.761,E2 -25059.761} C_VEL
LIN {X 0,Y 133.103,Z 468.857,A -85,B 0,C 180,E1 -25064.539,E2 -25064.539} C_VEL
LIN {X 0,Y 129.959,Z 471.654,A -85,B 0,C 180,E1 -25069.542,E2 -25069.542} C_VEL
LIN {X 0,Y 128.386,Z 472.858,A -85,B 0,C 180,E1 -25072.979,E2 -25072.979} C_VEL
LIN {X 0,Y 127.216,Z 473.563,A -85,B 0,C 180,E1 -25076.468,E2 -25076.468} C_VEL
LIN {X 0,Y 126.375,Z 473.816,A -85,B 0,C 180,E1 -25079.969,E2 -25079.969} C_VEL
LIN {X 0,Y 125.923,Z 473.547,A -85,B 0,C 180,E1 -25083.484,E2 -25083.484} C_VEL
LIN {X 0,Y 125.694,Z 472.834,A -85,B 0,C 180,E1 -25086.962,E2 -25086.962} C_VEL
LIN {X 0,Y 125.966,Z 471.19,A -85,B 0,C 180,E1 -25091.487,E2 -25091.487} C_VEL
LIN {X 0,Y 126.985,Z 467.878,A -85,B 0,C 180,E1 -25097.213,E2 -25097.213} C_VEL
LIN {X 0,Y 128.62,Z 463.58,A -85,B 0,C 180,E1 -25102.327,E2 -25102.327} C_VEL
LIN {X 0,Y 131.11,Z 457.352,A -85,B 0,C 180,E1 -25107.698,E2 -25107.698} C_VEL
LIN {X 0,Y 134.127,Z 450.428,A -85,B 0,C 180,E1 -25112.183,E2 -25112.183} C_VEL
LIN {X 0,Y 137.23,Z 443.104,A -85,B 0,C 180,E1 -25115.881,E2 -25115.881} C_VEL
LIN {X 0,Y 140.791,Z 434.377,A -85,B 0,C 180,E1 -25119.339,E2 -25119.339} C_VEL
LIN {X 0,Y 144.378,Z 424.837,A -85,B 0,C 180,E1 -25122.265,E2 -25122.265} C_VEL
LIN {X 0,Y 147.929,Z 414.161,A -85,B 0,C 180,E1 -25124.797,E2 -25124.797} C_VEL
LIN {X 0,Y 151.119,Z 402.644,A -85,B 0,C 180,E1 -25126.9,E2 -25126.9} C_VEL
LIN {X 0,Y 153.712,Z 390.945,A -85,B 0,C 180,E1 -25128.495,E2 -25128.495} C_VEL
LIN {X 0,Y 155.898,Z 378.151,A -85,B 0,C 180,E1 -25129.695,E2 -25129.695} C_VEL
LIN {X 0,Y 157.357,Z 365.196,A -85,B 0,C 180,E1 -25130.46,E2 -25130.46} C_VEL
LIN {X 0,Y 160.072,Z 325.576,A -85,B 0,C 180,E1 -25132.086,E2 -25132.086} C_VEL
LIN {X 0,Y 155.65,Z 314.034,A -85,B 0,C 180,E1 -25134.125,E2 -25134.125} C_VEL
LIN {X 0,Y 151.994,Z 306.501,A -85,B 0,C 180,E1 -25135.801,E2 -25135.801} C_VEL
LIN {X 0,Y 145.171,Z 294.925,A -85,B 0,C 180,E1 -25139.104,E2 -25139.104} C_VEL
LIN {X 0,Y 140.757,Z 288.192,A -85,B 0,C 180,E1 -25141.439,E2 -25141.439} C_VEL
LIN {X 0,Y 138.112,Z 284.368,A -85,B 0,C 180,E1 -25142.934,E2 -25142.934} C_VEL
LIN {X 0,Y 135.435,Z 280.5,A -85,B 0,C 180,E1 -25144.545,E2 -25144.545} C_VEL
LIN {X 0,Y 133.242,Z 277.683,A -85,B 0,C 180,E1 -25145.924,E2 -25145.924} C_VEL
LIN {X 0,Y 132.253,Z 276.064,A -85,B 0,C 180,E1 -25146.608,E2 -25146.608} C_VEL
LIN {X 0,Y 130.083,Z 273.94,A -85,B 0,C 180,E1 -25148.045,E2 -25148.045} C_VEL
LIN {X 0,Y 129.106,Z 271.585,A -85,B 0,C 180,E1 -25149.106,E2 -25149.106} C_VEL
LIN {X 0,Y 128.917,Z 270.959,A -85,B 0,C 180,E1 -25150.27,E2 -25150.27} C_VEL
LIN {X 0,Y 128.9,Z 270.909,A -85,B 0,C 180,E1 -25155.14,E2 -25155.14} C_VEL
LIN {X 0,Y 128.922,Z 270.887,A -85,B 0,C 180,E1 -25159.749,E2 -25159.749} C_VEL
LIN {X 0,Y 128.942,Z 270.909,A -85,B 0,C 180,E1 -25164.847,E2 -25164.847} C_VEL
LIN {X 0,Y 128.97,Z 270.867,A -85,B 0,C 180,E1 -25170.683,E2 -25170.683} C_VEL
LIN {X 0,Y 129.062,Z 270.901,A -85,B 0,C 180,E1 -25177.784,E2 -25177.784} C_VEL
LIN {X 0,Y 129.148,Z 270.845,A -85,B 0,C 180,E1 -25184.223,E2 -25184.223} C_VEL
LIN {X 0,Y 129.345,Z 270.872,A -85,B 0,C 180,E1 -25187.98,E2 -25187.98} C_VEL
LIN {X 0,Y 129.462,Z 270.827,A -85,B 0,C 180,E1 -25190.638,E2 -25190.638} C_VEL
LIN {X 0,Y 130.071,Z 270.781,A -85,B 0,C 180,E1 -25200.011,E2 -25200.011} C_VEL
LIN {X 0,Y 129.472,Z 270.847,A -85,B 0,C 180,E1 -25209.383,E2 -25209.383} C_VEL
LIN {X 0,Y 129.309,Z 270.851,A -85,B 0,C 180,E1 -25212.567,E2 -25212.567} C_VEL
LIN {X 0,Y 129.127,Z 270.891,A -85,B 0,C 180,E1 -25219.071,E2 -25219.071} C_VEL
LIN {X 0,Y 129.119,Z 270.872,A -85,B 0,C 180,E1 -25222.407,E2 -25222.407} C_VEL
LIN {X 0,Y 129.116,Z 271.149,A -85,B 0,C 180,E1 -25227.351,E2 -25227.351} C_VEL
LIN {X 0,Y 129.374,Z 272.227,A -85,B 0,C 180,E1 -25228.171,E2 -25228.171} C_VEL
LIN {X 0,Y 130.94,Z 274.895,A -85,B 0,C 180,E1 -25229.375,E2 -25229.375} C_VEL
LIN {X 0,Y 132.745,Z 276.562,A -85,B 0,C 180,E1 -25230.537,E2 -25230.537} C_VEL
LIN {X 0,Y 135.112,Z 280.13,A -85,B 0,C 180,E1 -25232.09,E2 -25232.09} C_VEL
LIN {X 0,Y 136.385,Z 281.724,A -85,B 0,C 180,E1 -25232.856,E2 -25232.856} C_VEL
LIN {X 0,Y 141.767,Z 289.677,A -85,B 0,C 180,E1 -25235.938,E2 -25235.938} C_VEL
LIN {X 0,Y 147.566,Z 299.103,A -85,B 0,C 180,E1 -25238.946,E2 -25238.946} C_VEL
LIN {X 0,Y 152.757,Z 310.354,A -85,B 0,C 180,E1 -25241.537,E2 -25241.537} C_VEL
LIN {X 0,Y 157.324,Z 322.056,A -85,B 0,C 180,E1 -25243.716,E2 -25243.716} C_VEL
LIN {X 0,Y 159.9,Z 329.321,A -85,B 0,C 180,E1 -25244.919,E2 -25244.919} C_VEL
LIN {X 0,Y 156.777,Z 374.114,A -85,B 0,C 180,E1 -25246.827,E2 -25246.827} C_VEL
LIN {X 0,Y 154.747,Z 387.95,A -85,B 0,C 180,E1 -25247.83,E2 -25247.83} C_VEL
LIN {X 0,Y 152.41,Z 399.702,A -85,B 0,C 180,E1 -25249.137,E2 -25249.137} C_VEL
LIN {X 0,Y 149.311,Z 411.676,A -85,B 0,C 180,E1 -25250.98,E2 -25250.98} C_VEL
LIN {X 0,Y 145.749,Z 423.176,A -85,B 0,C 180,E1 -25253.362,E2 -25253.362} C_VEL
LIN {X 0,Y 141.992,Z 433.54,A -85,B 0,C 180,E1 -25256.161,E2 -25256.161} C_VEL
LIN {X 0,Y 138.383,Z 442.854,A -85,B 0,C 180,E1 -25259.476,E2 -25259.476} C_VEL
LIN {X 0,Y 135.29,Z 450.532,A -85,B 0,C 180,E1 -25262.962,E2 -25262.962} C_VEL
LIN {X 0,Y 132.002,Z 458.025,A -85,B 0,C 180,E1 -25267.292,E2 -25267.292} C_VEL
LIN {X 0,Y 129.092,Z 464.906,A -85,B 0,C 180,E1 -25272.574,E2 -25272.574} C_VEL
LIN {X 0,Y 127.518,Z 469.43,A -85,B 0,C 180,E1 -25277.262,E2 -25277.262} C_VEL
LIN {X 0,Y 126.831,Z 471.805,A -85,B 0,C 180,E1 -25280.428,E2 -25280.428} C_VEL
LIN {X 0,Y 126.431,Z 473.741,A -85,B 0,C 180,E1 -25283.614,E2 -25283.614} C_VEL
LIN {X 0,Y 126.265,Z 475.242,A -85,B 0,C 180,E1 -25286.807,E2 -25286.807} C_VEL
LIN {X 0,Y 126.338,Z 476.286,A -85,B 0,C 180,E1 -25289.997,E2 -25289.997} C_VEL
LIN {X 0,Y 126.265,Z 476.928,A -85,B 0,C 180,E1 -25293.188,E2 -25293.188} C_VEL
LIN {X 0,Y 126.904,Z 477.061,A -85,B 0,C 180,E1 -25299.561,E2 -25299.561} C_VEL
LIN {X 0,Y 128.731,Z 475.585,A -85,B 0,C 180,E1 -25305.838,E2 -25305.838} C_VEL
LIN {X 0,Y 131.896,Z 472.565,A -85,B 0,C 180,E1 -25311.897,E2 -25311.897} C_VEL
LIN {X 0,Y 135.354,Z 469.15,A -85,B 0,C 180,E1 -25316.187,E2 -25316.187} C_VEL
LIN {X 0,Y 137.273,Z 467.092,A -85,B 0,C 180,E1 -25318.194,E2 -25318.194} C_VEL
LIN {X 0,Y 138.832,Z 464.773,A -85,B 0,C 180,E1 -25320.351,E2 -25320.351} C_VEL
LIN {X 0,Y 140.066,Z 460.686,A -85,B 0,C 180,E1 -25324.026,E2 -25324.026} C_VEL
LIN {X 0,Y 141.676,Z 456.089,A -85,B 0,C 180,E1 -25327.525,E2 -25327.525} C_VEL
LIN {X 0,Y 143.742,Z 452.844,A -85,B 0,C 180,E1 -25329.335,E2 -25329.335} C_VEL
LIN {X 0,Y 149.05,Z 445.719,A -85,B 0,C 180,E1 -25332.212,E2 -25332.212} C_VEL
LIN {X 0,Y 154.521,Z 437.383,A -85,B 0,C 180,E1 -25334.824,E2 -25334.824} C_VEL
LIN {X 0,Y 159.833,Z 428.266,A -85,B 0,C 180,E1 -25336.968,E2 -25336.968} C_VEL
LIN {X 0,Y 164.676,Z 418.426,A -85,B 0,C 180,E1 -25338.777,E2 -25338.777} C_VEL
LIN {X 0,Y 169.685,Z 406.101,A -85,B 0,C 180,E1 -25340.477,E2 -25340.477} C_VEL
LIN {X 0,Y 173.621,Z 393.595,A -85,B 0,C 180,E1 -25341.742,E2 -25341.742} C_VEL
LIN {X 0,Y 176.684,Z 380.517,A -85,B 0,C 180,E1 -25342.595,E2 -25342.595} C_VEL
LIN {X 0,Y 178.552,Z 367.6,A -85,B 0,C 180,E1 -25343.173,E2 -25343.173} C_VEL
LIN {X 0,Y 180.382,Z 347.47,A -85,B 0,C 180,E1 -25343.885,E2 -25343.885} C_VEL
LIN {X 0,Y 177.746,Z 340.246,A -85,B 0,C 180,E1 -25346.23,E2 -25346.23} C_VEL
LIN {X 0,Y 174.593,Z 332.754,A -85,B 0,C 180,E1 -25349.385,E2 -25349.385} C_VEL
LIN {X 0,Y 172.136,Z 327.555,A -85,B 0,C 180,E1 -25352.227,E2 -25352.227} C_VEL
LIN {X 0,Y 169.973,Z 323.946,A -85,B 0,C 180,E1 -25355.187,E2 -25355.187} C_VEL
LIN {X 0,Y 167.859,Z 320.458,A -85,B 0,C 180,E1 -25358.954,E2 -25358.954} C_VEL
LIN {X 0,Y 167.443,Z 319.76,A -85,B 0,C 180,E1 -25359.913,E2 -25359.913} C_VEL
LIN {X 0,Y 165.642,Z 316.954,A -85,B 0,C 180,E1 -25367.744,E2 -25367.744} C_VEL
LIN {X 0,Y 165.753,Z 316.865,A -85,B 0,C 180,E1 -25370.619,E2 -25370.619} C_VEL
LIN {X 0,Y 167.795,Z 319.558,A -85,B 0,C 180,E1 -25377.953,E2 -25377.953} C_VEL
LIN {X 0,Y 169.663,Z 323.166,A -85,B 0,C 180,E1 -25381.534,E2 -25381.534} C_VEL
LIN {X 0,Y 170.696,Z 324.659,A -85,B 0,C 180,E1 -25383.037,E2 -25383.037} C_VEL
LIN {X 0,Y 172.898,Z 328.593,A -85,B 0,C 180,E1 -25385.88,E2 -25385.88} C_VEL
LIN {X 0,Y 176.112,Z 334.393,A -85,B 0,C 180,E1 -25389.244,E2 -25389.244} C_VEL
LIN {X 0,Y 178.258,Z 338.879,A -85,B 0,C 180,E1 -25391.226,E2 -25391.226} C_VEL
LIN {X 0,Y 180.578,Z 344.986,A -85,B 0,C 180,E1 -25393.255,E2 -25393.255} C_VEL
LIN {X 0,Y 177.943,Z 371.598,A -85,B 0,C 180,E1 -25394.216,E2 -25394.216} C_VEL
LIN {X 0,Y 175.535,Z 384.386,A -85,B 0,C 180,E1 -25394.907,E2 -25394.907} C_VEL
LIN {X 0,Y 172.214,Z 396.881,A -85,B 0,C 180,E1 -25395.947,E2 -25395.947} C_VEL
LIN {X 0,Y 168.37,Z 408.095,A -85,B 0,C 180,E1 -25397.294,E2 -25397.294} C_VEL
LIN {X 0,Y 163.547,Z 419.221,A -85,B 0,C 180,E1 -25399.03,E2 -25399.03} C_VEL
LIN {X 0,Y 158.214,Z 429.469,A -85,B 0,C 180,E1 -25401.126,E2 -25401.126} C_VEL
LIN {X 0,Y 152.206,Z 439.339,A -85,B 0,C 180,E1 -25403.834,E2 -25403.834} C_VEL
LIN {X 0,Y 145.986,Z 448.069,A -85,B 0,C 180,E1 -25407.055,E2 -25407.055} C_VEL
LIN {X 0,Y 140.524,Z 454.896,A -85,B 0,C 180,E1 -25410.433,E2 -25410.433} C_VEL
LIN {X 0,Y 135.649,Z 460.369,A -85,B 0,C 180,E1 -25414.013,E2 -25414.013} C_VEL
LIN {X 0,Y 130.526,Z 465.595,A -85,B 0,C 180,E1 -25418.677,E2 -25418.677} C_VEL
LIN {X 0,Y 126.298,Z 469.453,A -85,B 0,C 180,E1 -25423.668,E2 -25423.668} C_VEL
LIN {X 0,Y 123.743,Z 471.495,A -85,B 0,C 180,E1 -25427.571,E2 -25427.571} C_VEL
LIN {X 0,Y 122.112,Z 472.673,A -85,B 0,C 180,E1 -25430.725,E2 -25430.725} C_VEL
LIN {X 0,Y 120.585,Z 473.559,A -85,B 0,C 180,E1 -25434.66,E2 -25434.66} C_VEL
LIN {X 0,Y 119.627,Z 473.877,A -85,B 0,C 180,E1 -25438.083,E2 -25438.083} C_VEL
LIN {X 0,Y 118.901,Z 473.711,A -85,B 0,C 180,E1 -25442.423,E2 -25442.423} C_VEL
LIN {X 0,Y 118.649,Z 473.183,A -85,B 0,C 180,E1 -25445.507,E2 -25445.507} C_VEL
LIN {X 0,Y 118.823,Z 471.392,A -85,B 0,C 180,E1 -25451.105,E2 -25451.105} C_VEL
LIN {X 0,Y 119.667,Z 468.618,A -85,B 0,C 180,E1 -25456.416,E2 -25456.416} C_VEL
LIN {X 0,Y 121.387,Z 464.235,A -85,B 0,C 180,E1 -25462.193,E2 -25462.193} C_VEL
LIN {X 0,Y 123.301,Z 459.584,A -85,B 0,C 180,E1 -25466.735,E2 -25466.735} C_VEL
LIN {X 0,Y 126.552,Z 452.494,A -85,B 0,C 180,E1 -25471.993,E2 -25471.993} C_VEL
LIN {X 0,Y 129.938,Z 444.945,A -85,B 0,C 180,E1 -25476.213,E2 -25476.213} C_VEL
LIN {X 0,Y 133.518,Z 436.581,A -85,B 0,C 180,E1 -25479.852,E2 -25479.852} C_VEL
LIN {X 0,Y 137.628,Z 426.435,A -85,B 0,C 180,E1 -25483.243,E2 -25483.243} C_VEL
LIN {X 0,Y 141.325,Z 416.11,A -85,B 0,C 180,E1 -25485.876,E2 -25485.876} C_VEL
LIN {X 0,Y 144.633,Z 405.017,A -85,B 0,C 180,E1 -25488.048,E2 -25488.048} C_VEL
LIN {X 0,Y 147.53,Z 392.851,A -85,B 0,C 180,E1 -25489.844,E2 -25489.844} C_VEL
